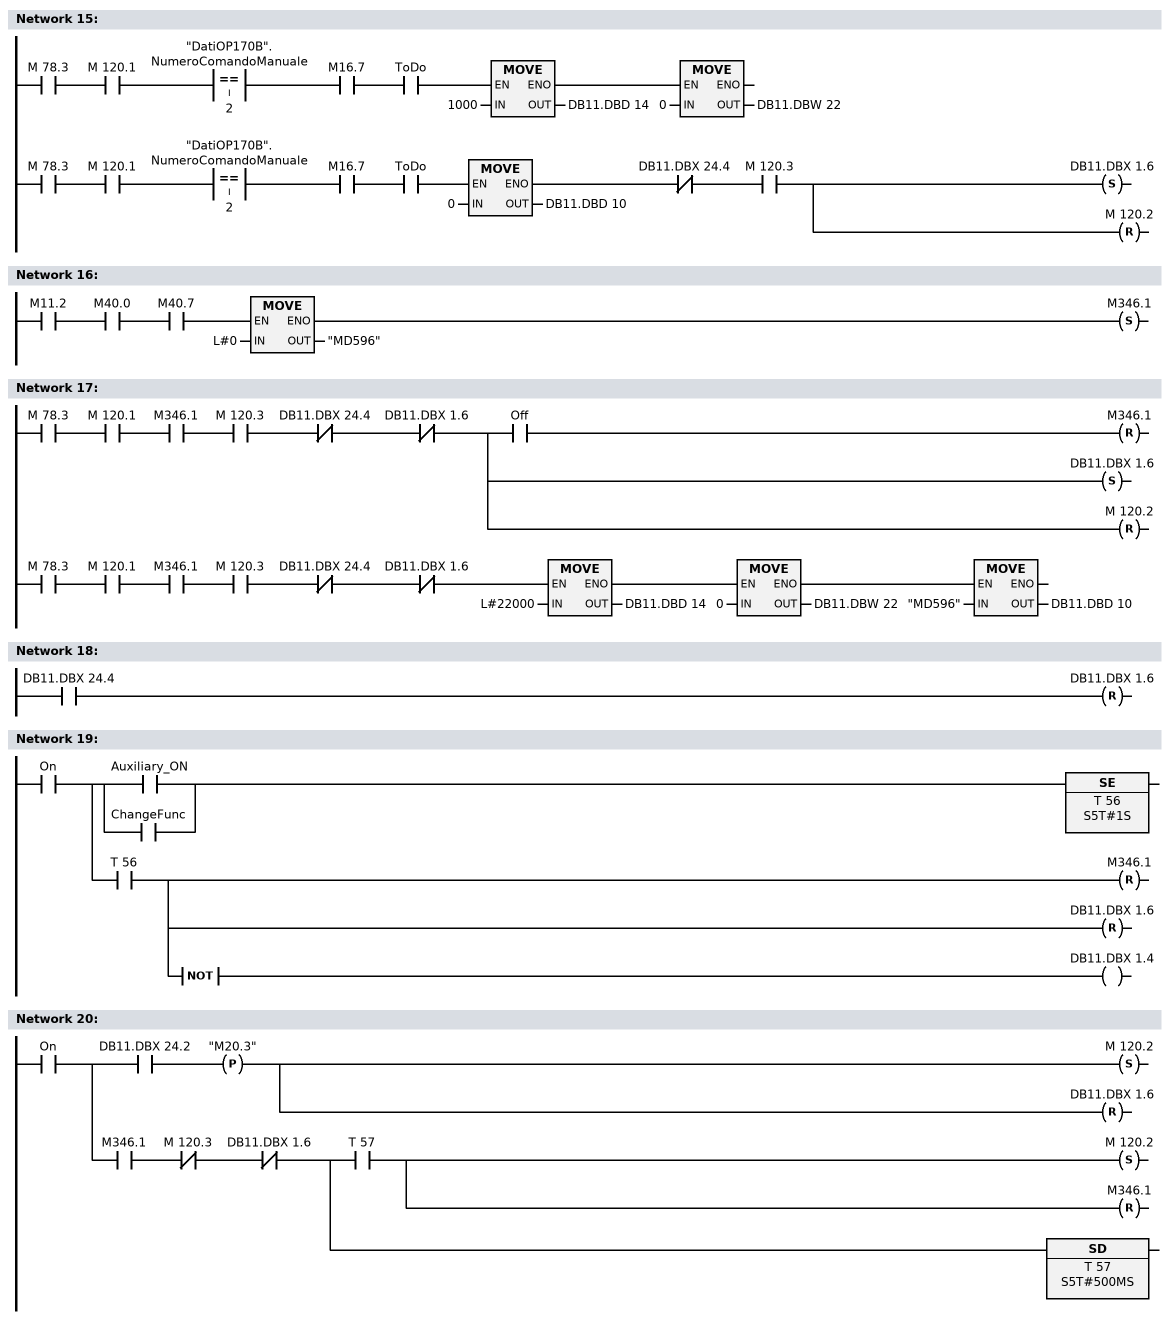
[picture p48: FC - AUTOMATIC networks 15-20]
NETWORK
TITLE =
      A     M 78.3;
      A     M 120.1;
      A(;
      L     "DatiOP170B".NumeroComandoManuale;
      L     2;
      ==I;
      );
      A     "M16.7";
      =     L 21.0;
      A(;
      A     L 21.0;
      A     "ToDo";
      JNB   M012;
      L     1000;
      T     DB11.DBD 14;
      SET;
      SAVE;
      CLR;
M012: A     BR;
      );
      JNB   M013;
      L     0;
      T     DB11.DBW 22;
M013: NOP   0;
      A(;
      A     L 21.0;
      A     "ToDo";
      JNB   M014;
      L     0;
      T     DB11.DBD 10;
      SET;
      SAVE;
      CLR;
M014: A     BR;
      );
      AN    DB11.DBX 24.4;
      A     M 120.3;
      S     DB11.DBX 1.6;
      R     M 120.2;
NETWORK
TITLE =
      A     "M11.2";
      A     "M40.0";
      A     "M40.7";
      JNB   M015;
      L     L#0;
      T     "MD596";
      SET;
      SAVE;
      CLR;
M015: A     BR;
      S     "M346.1";
NETWORK
TITLE =
      A     M 78.3;
      A     M 120.1;
      A     "M346.1";
      A     M 120.3;
      AN    DB11.DBX 24.4;
      AN    DB11.DBX 1.6;
      =     L 21.0;
      A(;
      A(;
      A     L 21.0;
      JNB   M016;
      L     L#22000;
      T     DB11.DBD 14;
      SET;
      SAVE;
      CLR;
M016: A     BR;
      );
      JNB   M017;
      L     0;
      T     DB11.DBW 22;
      SET;
      SAVE;
      CLR;
M017: A     BR;
      );
      JNB   M018;
      L     "MD596";
      T     DB11.DBD 10;
M018: NOP   0;
      A     L 21.0;
      A     "Off";
      R     "M346.1";
      A     L 21.0;
      BLD   102;
      S     DB11.DBX 1.6;
      A     L 21.0;
      BLD   102;
      R     M 120.2;
NETWORK
TITLE =
      A     DB11.DBX 24.4;
      R     DB11.DBX 1.6;
NETWORK
TITLE =
      A     "On";
      =     L 21.0;
      A     L 21.0;
      A(;
      O     "Auxiliary_ON";
      O     "ChangeFunc";
      );
      L     S5T#1S;
      SE    T 56;
      A     L 21.0;
      A     T 56;
      =     L 21.1;
      A     L 21.1;
      BLD   102;
      R     "M346.1";
      A     L 21.1;
      BLD   102;
      R     DB11.DBX 1.6;
      A     L 21.1;
      NOT;
      =     DB11.DBX 1.4;
NETWORK
TITLE =
      A     "On";
      =     L 21.0;
      A     L 21.0;
      A     DB11.DBX 24.2;
      FP    "M20.3";
      S     M 120.2;
      R     DB11.DBX 1.6;
      A     L 21.0;
      A     "M346.1";
      AN    M 120.3;
      AN    DB11.DBX 1.6;
      =     L 21.1;
      A     L 21.1;
      A     T 57;
      S     M 120.2;
      R     "M346.1";
      A     L 21.1;
      BLD   102;
      L     S5T#500MS;
      SD    T 57;
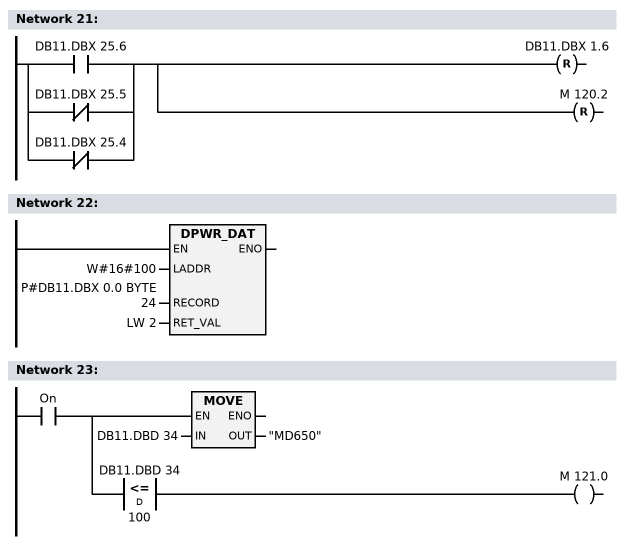
NETWORK
TITLE =
      O     DB11.DBX 25.6;
      ON    DB11.DBX 25.5;
      ON    DB11.DBX 25.4;
      R     DB11.DBX 1.6;
      R     M 120.2;
NETWORK
TITLE =
      CALL  "DPWR_DAT" (
           LADDR                    := W#16#100,
           RECORD                   := P#DB11.DBX 0.0 BYTE 24,
           RET_VAL                  := LW 2);
      NOP   0;
NETWORK
TITLE =
      A     "On";
      =     L 20.0;
      A     L 20.0;
      JNB   M019;
      L     DB11.DBD 34;
      T     "MD650";
M019: NOP   0;
      A     L 20.0;
      A(;
      L     DB11.DBD 34;
      L     100;
      <=D;
      );
      =     M 121.0;
END_FUNCTION

FUNCTION FC 25 : VOID
VERSION : 0.1
BEGIN
// (block stored without names or comments; labels and parameter names are numbered)
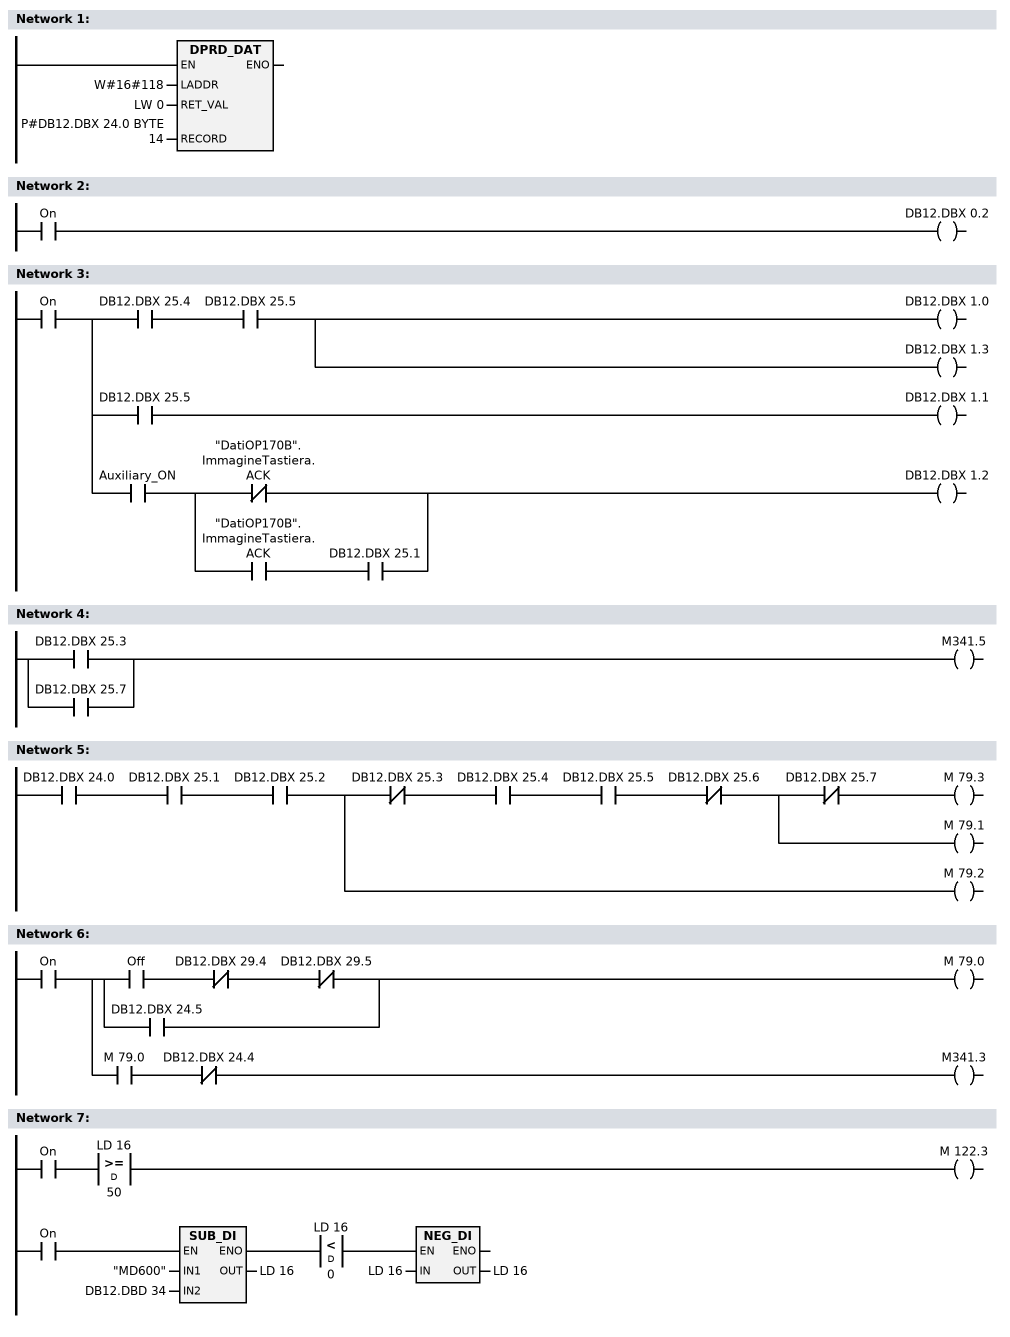
NETWORK
TITLE =
      CALL  "DPRD_DAT" (
           LADDR                    := W#16#118,
           RET_VAL                  := LW 0,
           RECORD                   := P#DB12.DBX 24.0 BYTE 14);
      NOP   0;
NETWORK
TITLE =
      A     "On";
      =     DB12.DBX 0.2;
NETWORK
TITLE =
      A     "On";
      =     L 21.0;
      A     L 21.0;
      A     DB12.DBX 25.4;
      A     DB12.DBX 25.5;
      =     DB12.DBX 1.0;
      =     DB12.DBX 1.3;
      A     L 21.0;
      A     DB12.DBX 25.5;
      =     DB12.DBX 1.1;
      A     L 21.0;
      A     "Auxiliary_ON";
      A(;
      ON    "DatiOP170B".ImmagineTastiera.ACK;
      O;
      A     "DatiOP170B".ImmagineTastiera.ACK;
      A     DB12.DBX 25.1;
      );
      =     DB12.DBX 1.2;
NETWORK
TITLE =
      O     DB12.DBX 25.3;
      O     DB12.DBX 25.7;
      =     "M341.5";
NETWORK
TITLE =
      A     DB12.DBX 24.0;
      A     DB12.DBX 25.1;
      A     DB12.DBX 25.2;
      =     L 21.0;
      A     L 21.0;
      AN    DB12.DBX 25.3;
      A     DB12.DBX 25.4;
      A     DB12.DBX 25.5;
      AN    DB12.DBX 25.6;
      =     L 21.1;
      A     L 21.1;
      AN    DB12.DBX 25.7;
      =     M 79.3;
      A     L 21.1;
      BLD   102;
      =     M 79.1;
      A     L 21.0;
      BLD   102;
      =     M 79.2;
NETWORK
TITLE =
      A     "On";
      =     L 21.0;
      A     L 21.0;
      A(;
      A     "Off";
      AN    DB12.DBX 29.4;
      AN    DB12.DBX 29.5;
      O     DB12.DBX 24.5;
      );
      =     M 79.0;
      A     L 21.0;
      A     M 79.0;
      AN    DB12.DBX 24.4;
      =     "M341.3";
NETWORK
TITLE =
      A     "On";
      =     L 20.0;
      A(;
      A     L 20.0;
      JNB   M001;
      L     "MD600";
      L     DB12.DBD 34;
      -D;
      T     LD 16;
      AN    OV;
      SAVE;
      CLR;
M001: A     BR;
      );
      A(;
      L     LD 16;
      L     0;
      <D;
      );
      JNB   M002;
      L     LD 16;
      NEGD;
      T     LD 16;
M002: NOP   0;
      A     L 20.0;
      A(;
      L     LD 16;
      L     50;
      >=D;
      );
      =     M 122.3;
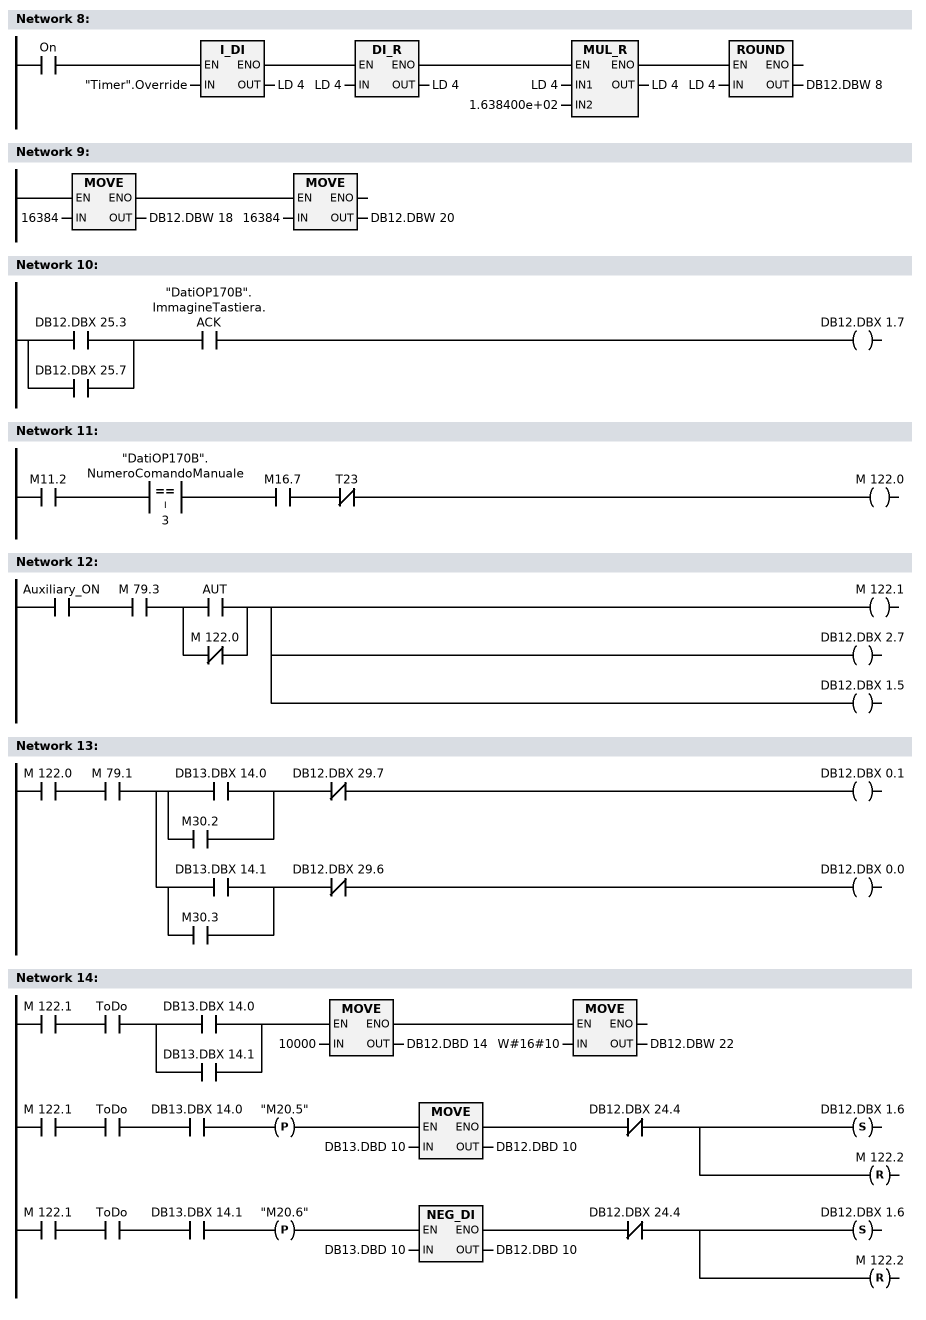
NETWORK
TITLE =
      A(;
      A(;
      A(;
      A     "On";
      JNB   M003;
      L     "Timer".Override;
      ITD;
      T     LD 4;
      SET;
      SAVE;
      CLR;
M003: A     BR;
      );
      JNB   M004;
      L     LD 4;
      DTR;
      T     LD 4;
      SET;
      SAVE;
      CLR;
M004: A     BR;
      );
      JNB   M005;
      L     LD 4;
      L     1.638400e+02;
      *R;
      T     LD 4;
      AN    OV;
      SAVE;
      CLR;
M005: A     BR;
      );
      JNB   M006;
      L     LD 4;
      RND;
      T     DB12.DBW 8;
M006: NOP   0;
NETWORK
TITLE =
      A(;
      L     16384;
      T     DB12.DBW 18;
      SET;
      SAVE;
      CLR;
      A     BR;
      );
      JNB   M007;
      L     16384;
      T     DB12.DBW 20;
M007: NOP   0;
NETWORK
TITLE =
      A(;
      O     DB12.DBX 25.3;
      O     DB12.DBX 25.7;
      );
      A     "DatiOP170B".ImmagineTastiera.ACK;
      =     DB12.DBX 1.7;
NETWORK
TITLE =
      A     "M11.2";
      A(;
      L     "DatiOP170B".NumeroComandoManuale;
      L     3;
      ==I;
      );
      A     "M16.7";
      AN    "T23";
      =     M 122.0;
NETWORK
TITLE =
      A     "Auxiliary_ON";
      A     M 79.3;
      A(;
      O     "AUT";
      ON    M 122.0;
      );
      =     M 122.1;
      =     DB12.DBX 2.7;
      =     DB12.DBX 1.5;
NETWORK
TITLE =
      A     M 122.0;
      A     M 79.1;
      =     L 21.0;
      A     L 21.0;
      A(;
      O     DB13.DBX 14.0;
      O     "M30.2";
      );
      AN    DB12.DBX 29.7;
      =     DB12.DBX 0.1;
      A     L 21.0;
      A(;
      O     DB13.DBX 14.1;
      O     "M30.3";
      );
      AN    DB12.DBX 29.6;
      =     DB12.DBX 0.0;
NETWORK
TITLE =
      A     M 122.1;
      A     "ToDo";
      =     L 21.0;
      A(;
      A     L 21.0;
      A(;
      O     DB13.DBX 14.0;
      O     DB13.DBX 14.1;
      );
      JNB   M008;
      L     10000;
      T     DB12.DBD 14;
      SET;
      SAVE;
      CLR;
M008: A     BR;
      );
      JNB   M009;
      L     W#16#10;
      T     DB12.DBW 22;
M009: NOP   0;
      A(;
      A     L 21.0;
      A     DB13.DBX 14.0;
      FP    "M20.5";
      JNB   M010;
      L     DB13.DBD 10;
      T     DB12.DBD 10;
      SET;
      SAVE;
      CLR;
M010: A     BR;
      );
      AN    DB12.DBX 24.4;
      S     DB12.DBX 1.6;
      R     M 122.2;
      A(;
      A     L 21.0;
      A     DB13.DBX 14.1;
      FP    "M20.6";
      JNB   M011;
      L     DB13.DBD 10;
      NEGD;
      T     DB12.DBD 10;
      AN    OV;
      SAVE;
      CLR;
M011: A     BR;
      );
      AN    DB12.DBX 24.4;
      S     DB12.DBX 1.6;
      R     M 122.2;
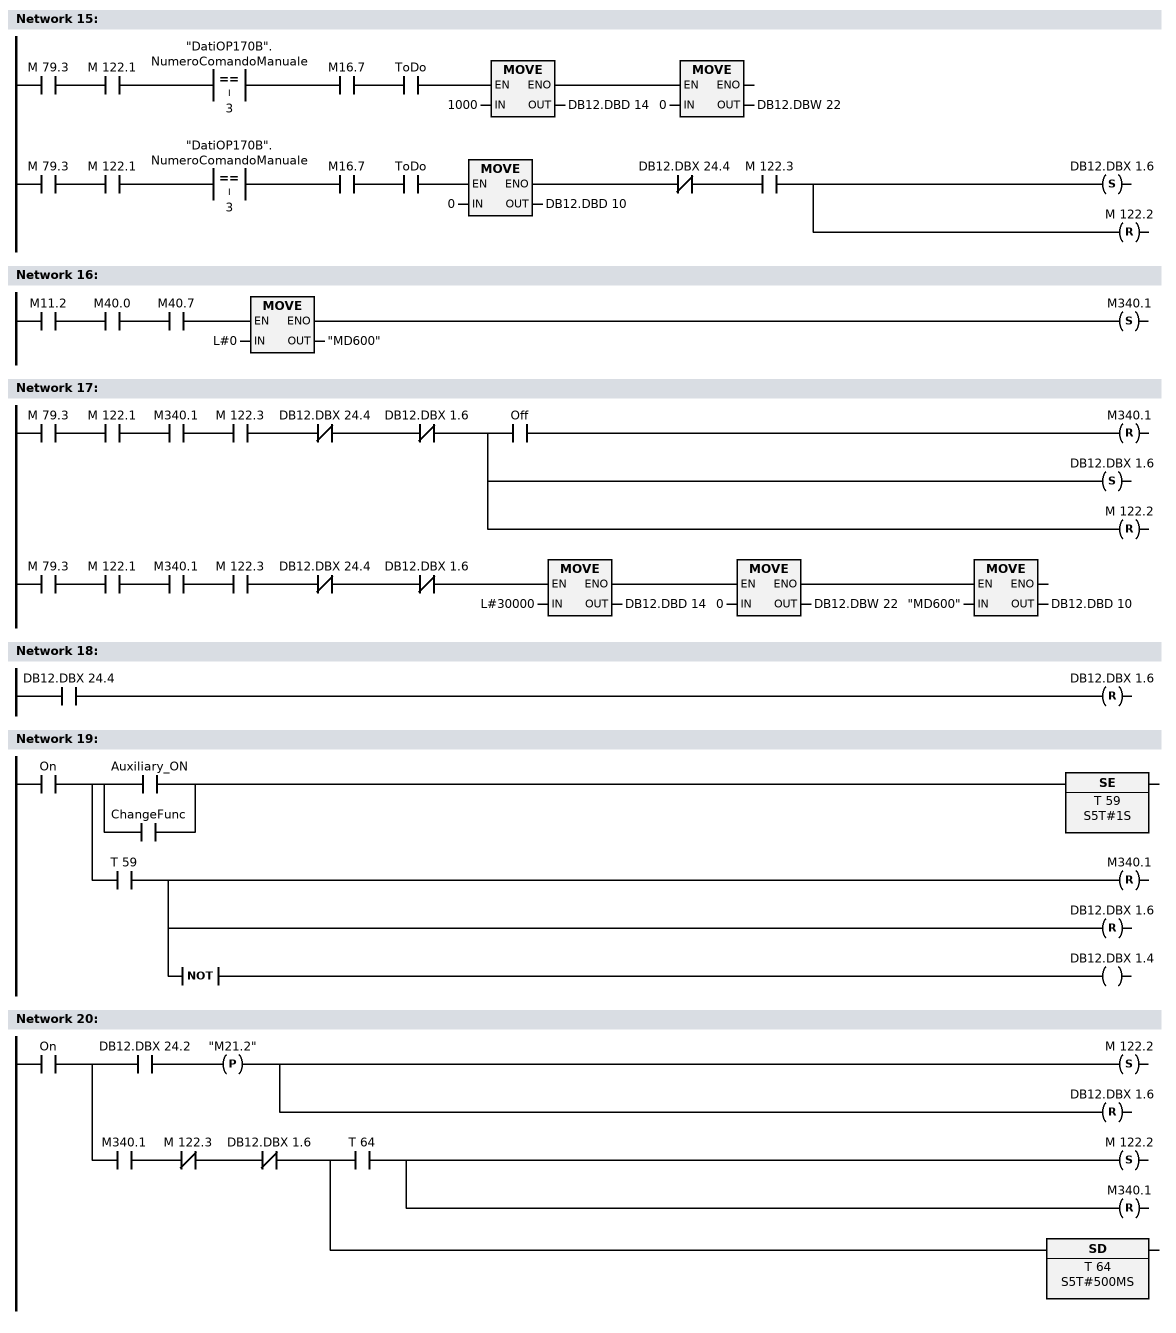
NETWORK
TITLE =
      A     M 79.3;
      A     M 122.1;
      A(;
      L     "DatiOP170B".NumeroComandoManuale;
      L     3;
      ==I;
      );
      A     "M16.7";
      =     L 21.0;
      A(;
      A     L 21.0;
      A     "ToDo";
      JNB   M012;
      L     1000;
      T     DB12.DBD 14;
      SET;
      SAVE;
      CLR;
M012: A     BR;
      );
      JNB   M013;
      L     0;
      T     DB12.DBW 22;
M013: NOP   0;
      A(;
      A     L 21.0;
      A     "ToDo";
      JNB   M014;
      L     0;
      T     DB12.DBD 10;
      SET;
      SAVE;
      CLR;
M014: A     BR;
      );
      AN    DB12.DBX 24.4;
      A     M 122.3;
      S     DB12.DBX 1.6;
      R     M 122.2;
NETWORK
TITLE =
      A     "M11.2";
      A     "M40.0";
      A     "M40.7";
      JNB   M015;
      L     L#0;
      T     "MD600";
      SET;
      SAVE;
      CLR;
M015: A     BR;
      S     "M340.1";
NETWORK
TITLE =
      A     M 79.3;
      A     M 122.1;
      A     "M340.1";
      A     M 122.3;
      AN    DB12.DBX 24.4;
      AN    DB12.DBX 1.6;
      =     L 21.0;
      A(;
      A(;
      A     L 21.0;
      JNB   M016;
      L     L#30000;
      T     DB12.DBD 14;
      SET;
      SAVE;
      CLR;
M016: A     BR;
      );
      JNB   M017;
      L     0;
      T     DB12.DBW 22;
      SET;
      SAVE;
      CLR;
M017: A     BR;
      );
      JNB   M018;
      L     "MD600";
      T     DB12.DBD 10;
M018: NOP   0;
      A     L 21.0;
      A     "Off";
      R     "M340.1";
      A     L 21.0;
      BLD   102;
      S     DB12.DBX 1.6;
      A     L 21.0;
      BLD   102;
      R     M 122.2;
NETWORK
TITLE =
      A     DB12.DBX 24.4;
      R     DB12.DBX 1.6;
NETWORK
TITLE =
      A     "On";
      =     L 21.0;
      A     L 21.0;
      A(;
      O     "Auxiliary_ON";
      O     "ChangeFunc";
      );
      L     S5T#1S;
      SE    T 59;
      A     L 21.0;
      A     T 59;
      =     L 21.1;
      A     L 21.1;
      BLD   102;
      R     "M340.1";
      A     L 21.1;
      BLD   102;
      R     DB12.DBX 1.6;
      A     L 21.1;
      NOT;
      =     DB12.DBX 1.4;
NETWORK
TITLE =
      A     "On";
      =     L 21.0;
      A     L 21.0;
      A     DB12.DBX 24.2;
      FP    "M21.2";
      S     M 122.2;
      R     DB12.DBX 1.6;
      A     L 21.0;
      A     "M340.1";
      AN    M 122.3;
      AN    DB12.DBX 1.6;
      =     L 21.1;
      A     L 21.1;
      A     T 64;
      S     M 122.2;
      R     "M340.1";
      A     L 21.1;
      BLD   102;
      L     S5T#500MS;
      SD    T 64;
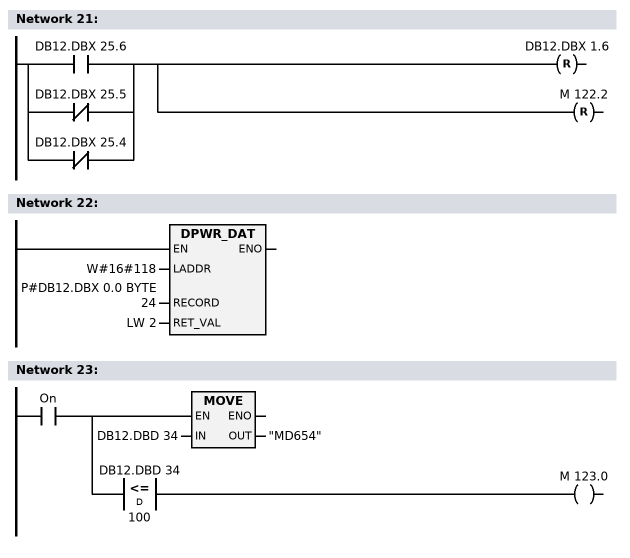
NETWORK
TITLE =
      O     DB12.DBX 25.6;
      ON    DB12.DBX 25.5;
      ON    DB12.DBX 25.4;
      R     DB12.DBX 1.6;
      R     M 122.2;
NETWORK
TITLE =
      CALL  "DPWR_DAT" (
           LADDR                    := W#16#118,
           RECORD                   := P#DB12.DBX 0.0 BYTE 24,
           RET_VAL                  := LW 2);
      NOP   0;
NETWORK
TITLE =
      A     "On";
      =     L 20.0;
      A     L 20.0;
      JNB   M019;
      L     DB12.DBD 34;
      T     "MD654";
M019: NOP   0;
      A     L 20.0;
      A(;
      L     DB12.DBD 34;
      L     100;
      <=D;
      );
      =     M 123.0;
END_FUNCTION

FUNCTION "FC50 - TEACH-IN" : VOID	// FC 50
VERSION : 0.1
VAR_TEMP
  TEMP0 : DINT ;
  TEMP1 : DINT ;
END_VAR
BEGIN
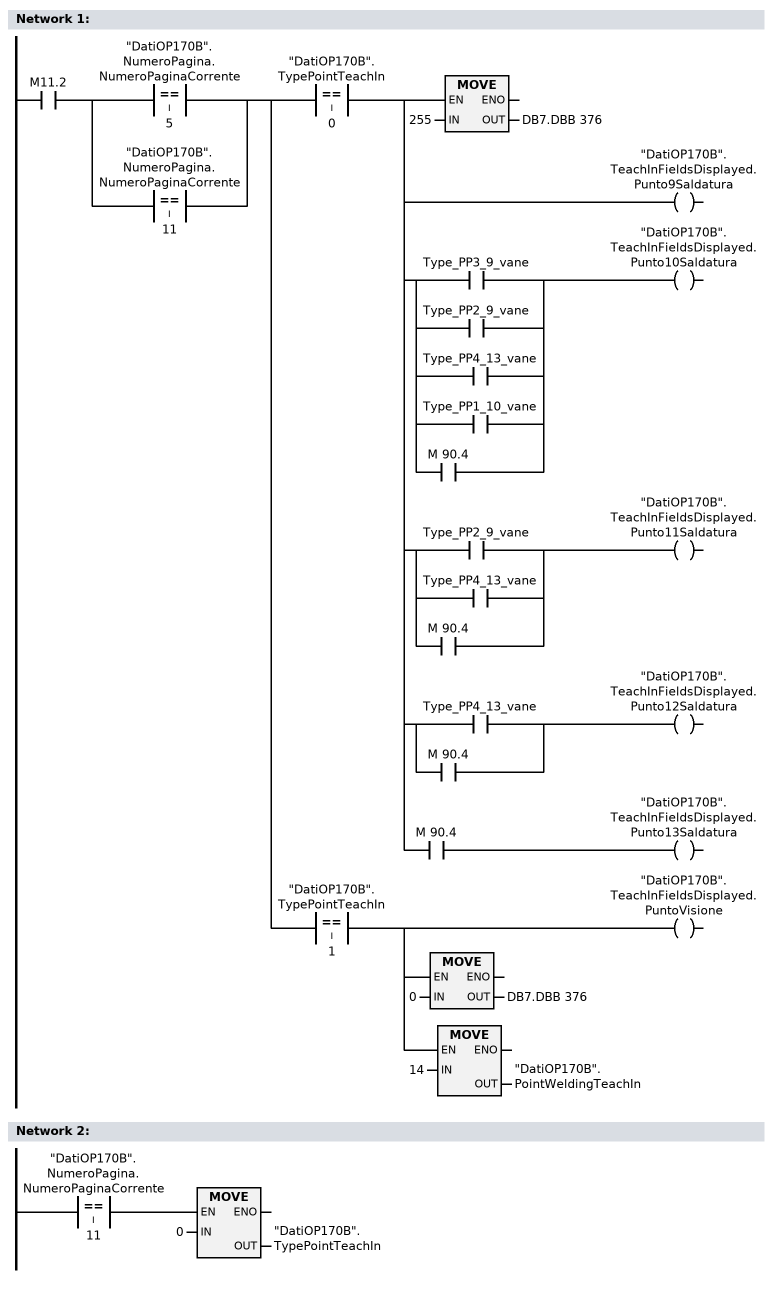
NETWORK
TITLE =
      A     "M11.2";
      A(;
      O(;
      L     "DatiOP170B".NumeroPagina.NumeroPaginaCorrente;
      L     5;
      ==I;
      );
      O(;
      L     "DatiOP170B".NumeroPagina.NumeroPaginaCorrente;
      L     11;
      ==I;
      );
      );
      =     L 8.0;
      A     L 8.0;
      A(;
      L     "DatiOP170B".TypePointTeachIn;
      L     0;
      ==I;
      );
      =     L 8.1;
      A     L 8.1;
      JNB   _001;
      L     255;
      T     DB7.DBB 376;
_001: NOP   0;
      A     L 8.1;
      BLD   102;
      =     "DatiOP170B".TeachInFieldsDisplayed.Punto9Saldatura;
      A     L 8.1;
      A(;
      O     "Type_PP3_9_vane";
      O     "Type_PP2_9_vane";
      O     "Type_PP4_13_vane";
      O     "Type_PP1_10_vane";
      O     M 90.4;
      );
      =     "DatiOP170B".TeachInFieldsDisplayed.Punto10Saldatura;
      A     L 8.1;
      A(;
      O     "Type_PP2_9_vane";
      O     "Type_PP4_13_vane";
      O     M 90.4;
      );
      =     "DatiOP170B".TeachInFieldsDisplayed.Punto11Saldatura;
      A     L 8.1;
      A(;
      O     "Type_PP4_13_vane";
      O     M 90.4;
      );
      =     "DatiOP170B".TeachInFieldsDisplayed.Punto12Saldatura;
      A     L 8.1;
      A     M 90.4;
      =     "DatiOP170B".TeachInFieldsDisplayed.Punto13Saldatura;
      A     L 8.0;
      A(;
      L     "DatiOP170B".TypePointTeachIn;
      L     1;
      ==I;
      );
      =     L 8.1;
      A     L 8.1;
      BLD   102;
      =     "DatiOP170B".TeachInFieldsDisplayed.PuntoVisione;
      A     L 8.1;
      JNB   _002;
      L     0;
      T     DB7.DBB 376;
_002: NOP   0;
      A     L 8.1;
      JNB   _003;
      L     14;
      T     "DatiOP170B".PointWeldingTeachIn;
_003: NOP   0;
NETWORK
TITLE =
      A(;
      L     "DatiOP170B".NumeroPagina.NumeroPaginaCorrente;
      L     11;
      ==I;
      );
      JNB   _004;
      L     0;
      T     "DatiOP170B".TypePointTeachIn;
_004: NOP   0;
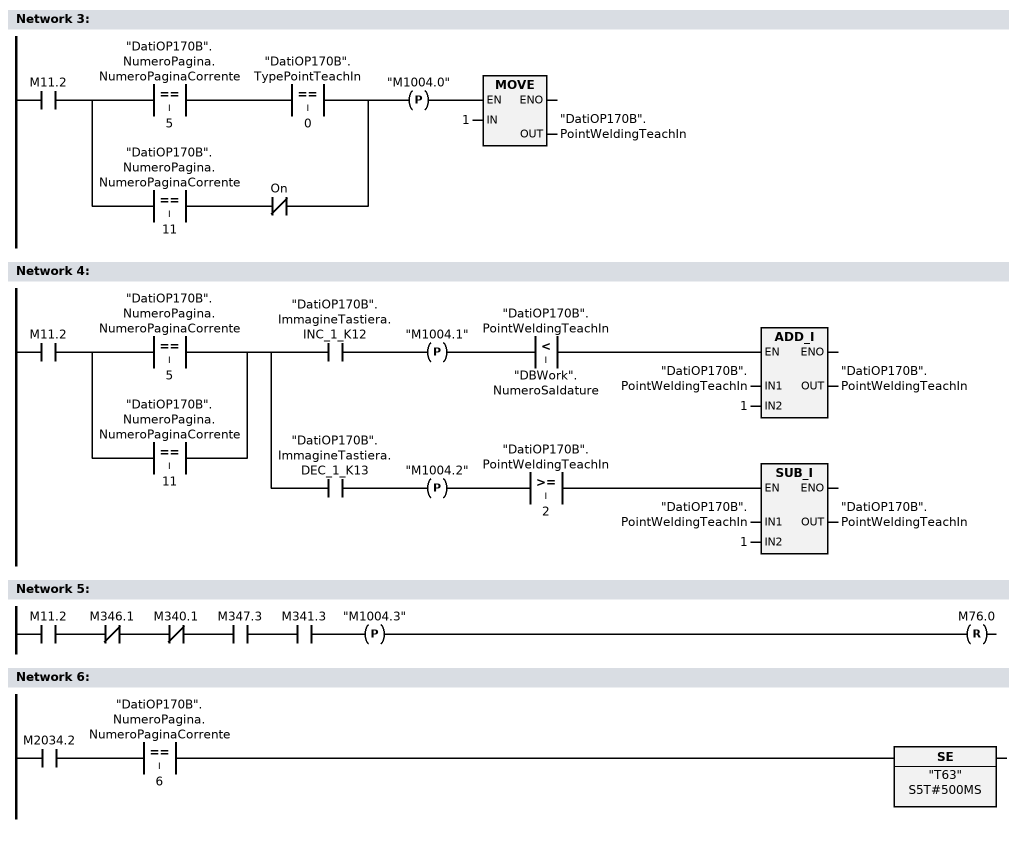
NETWORK
TITLE =
      A     "M11.2";
      A(;
      A(;
      L     "DatiOP170B".NumeroPagina.NumeroPaginaCorrente;
      L     5;
      ==I;
      );
      A(;
      L     "DatiOP170B".TypePointTeachIn;
      L     0;
      ==I;
      );
      O;
      A(;
      L     "DatiOP170B".NumeroPagina.NumeroPaginaCorrente;
      L     11;
      ==I;
      );
      AN    "On";
      );
      FP    "M1004.0";
      JNB   _005;
      L     1;
      T     "DatiOP170B".PointWeldingTeachIn;
_005: NOP   0;
NETWORK
TITLE =
      A     "M11.2";
      A(;
      O(;
      L     "DatiOP170B".NumeroPagina.NumeroPaginaCorrente;
      L     5;
      ==I;
      );
      O(;
      L     "DatiOP170B".NumeroPagina.NumeroPaginaCorrente;
      L     11;
      ==I;
      );
      );
      =     L 8.0;
      A     L 8.0;
      A     "DatiOP170B".ImmagineTastiera.INC_1_K12;
      FP    "M1004.1";
      A(;
      L     "DatiOP170B".PointWeldingTeachIn;
      L     "DBWork".NumeroSaldature;
      <I;
      );
      JNB   _006;
      L     "DatiOP170B".PointWeldingTeachIn;
      L     1;
      +I;
      T     "DatiOP170B".PointWeldingTeachIn;
_006: NOP   0;
      A     L 8.0;
      A     "DatiOP170B".ImmagineTastiera.DEC_1_K13;
      FP    "M1004.2";
      A(;
      L     "DatiOP170B".PointWeldingTeachIn;
      L     2;
      >=I;
      );
      JNB   _007;
      L     "DatiOP170B".PointWeldingTeachIn;
      L     1;
      -I;
      T     "DatiOP170B".PointWeldingTeachIn;
_007: NOP   0;
NETWORK
TITLE =
      A     "M11.2";
      AN    "M346.1";
      AN    "M340.1";
      A     "M347.3";
      A     "M341.3";
      FP    "M1004.3";
      R     "M76.0";
NETWORK
TITLE =
      A     "M2034.2";
      A(;
      L     "DatiOP170B".NumeroPagina.NumeroPaginaCorrente;
      L     6;
      ==I;
      );
      L     S5T#500MS;
      SE    "T63";
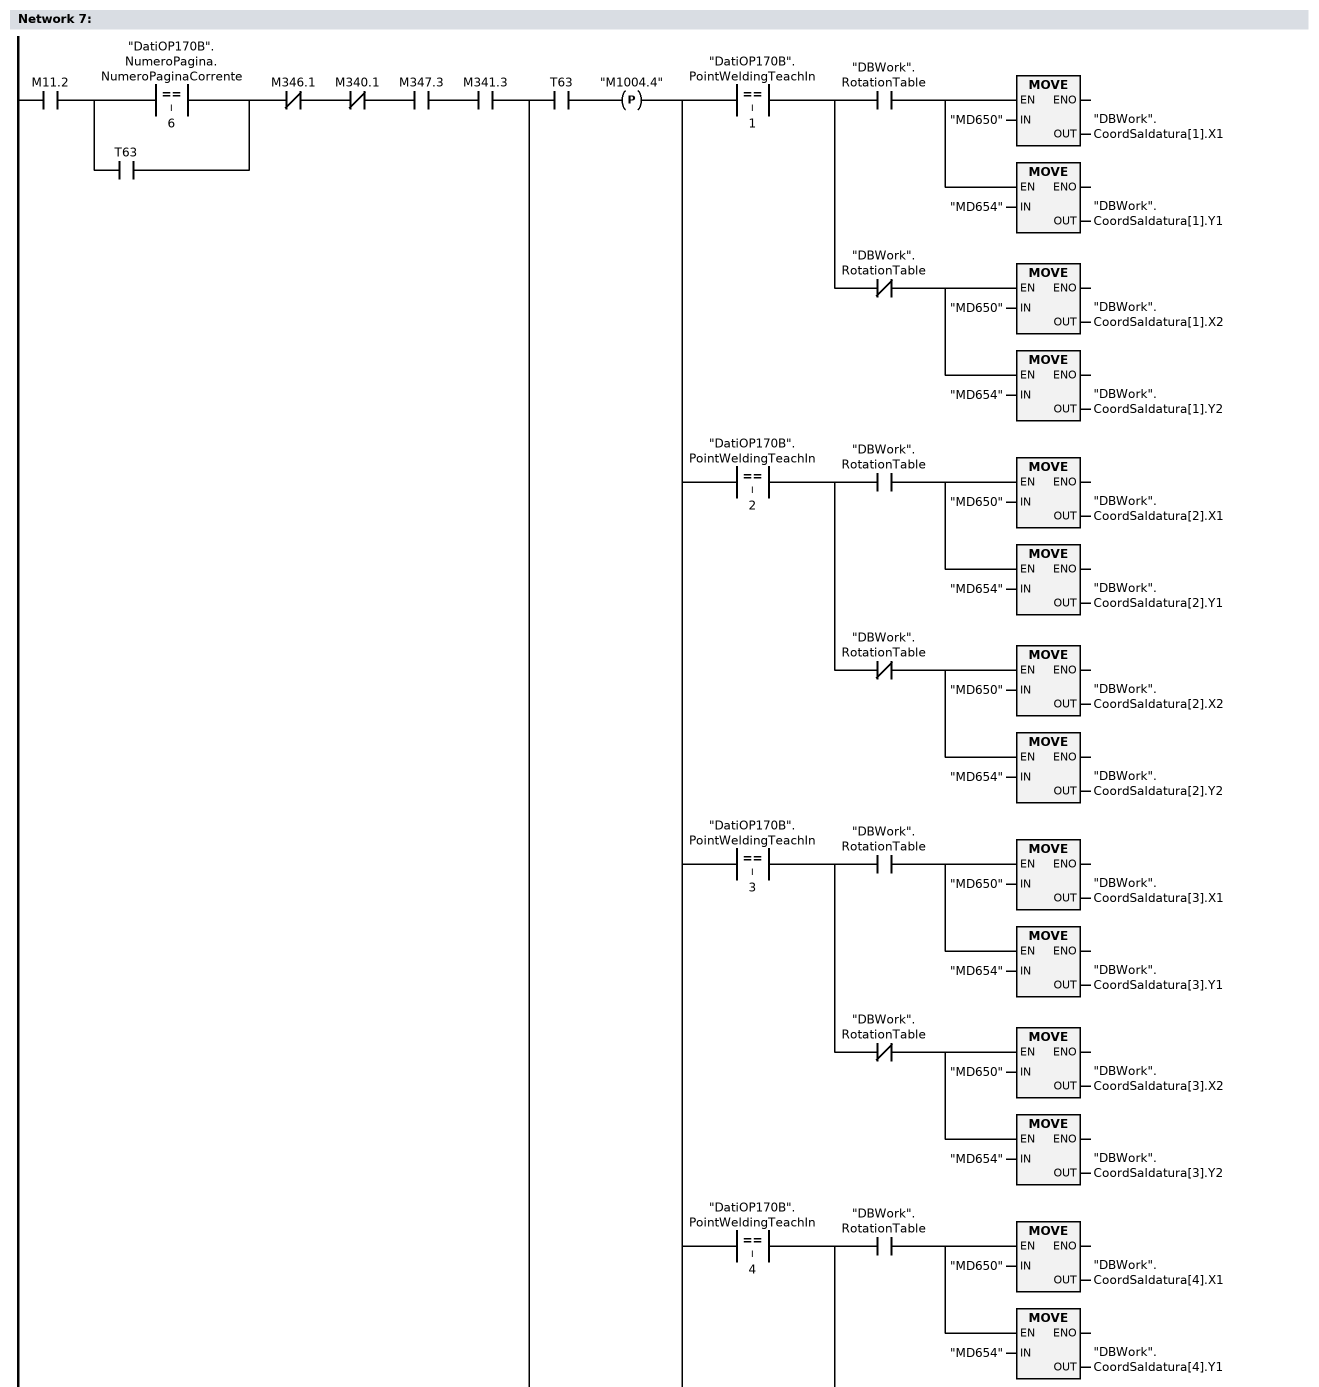
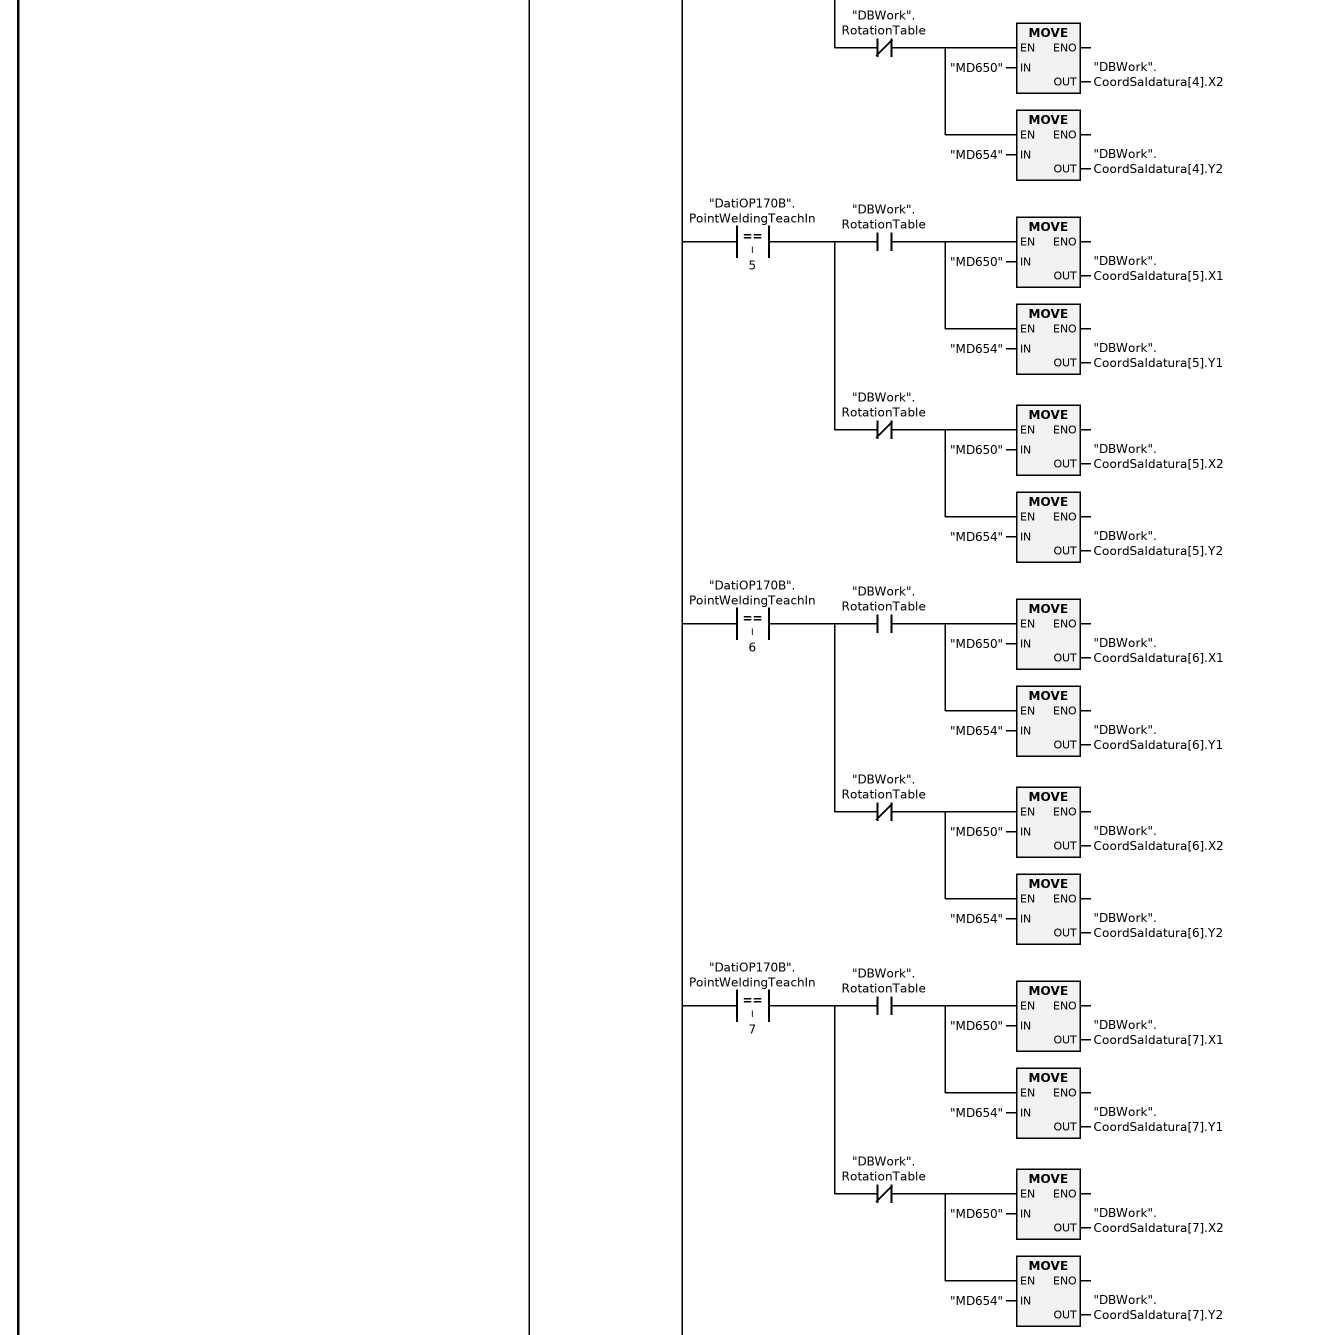
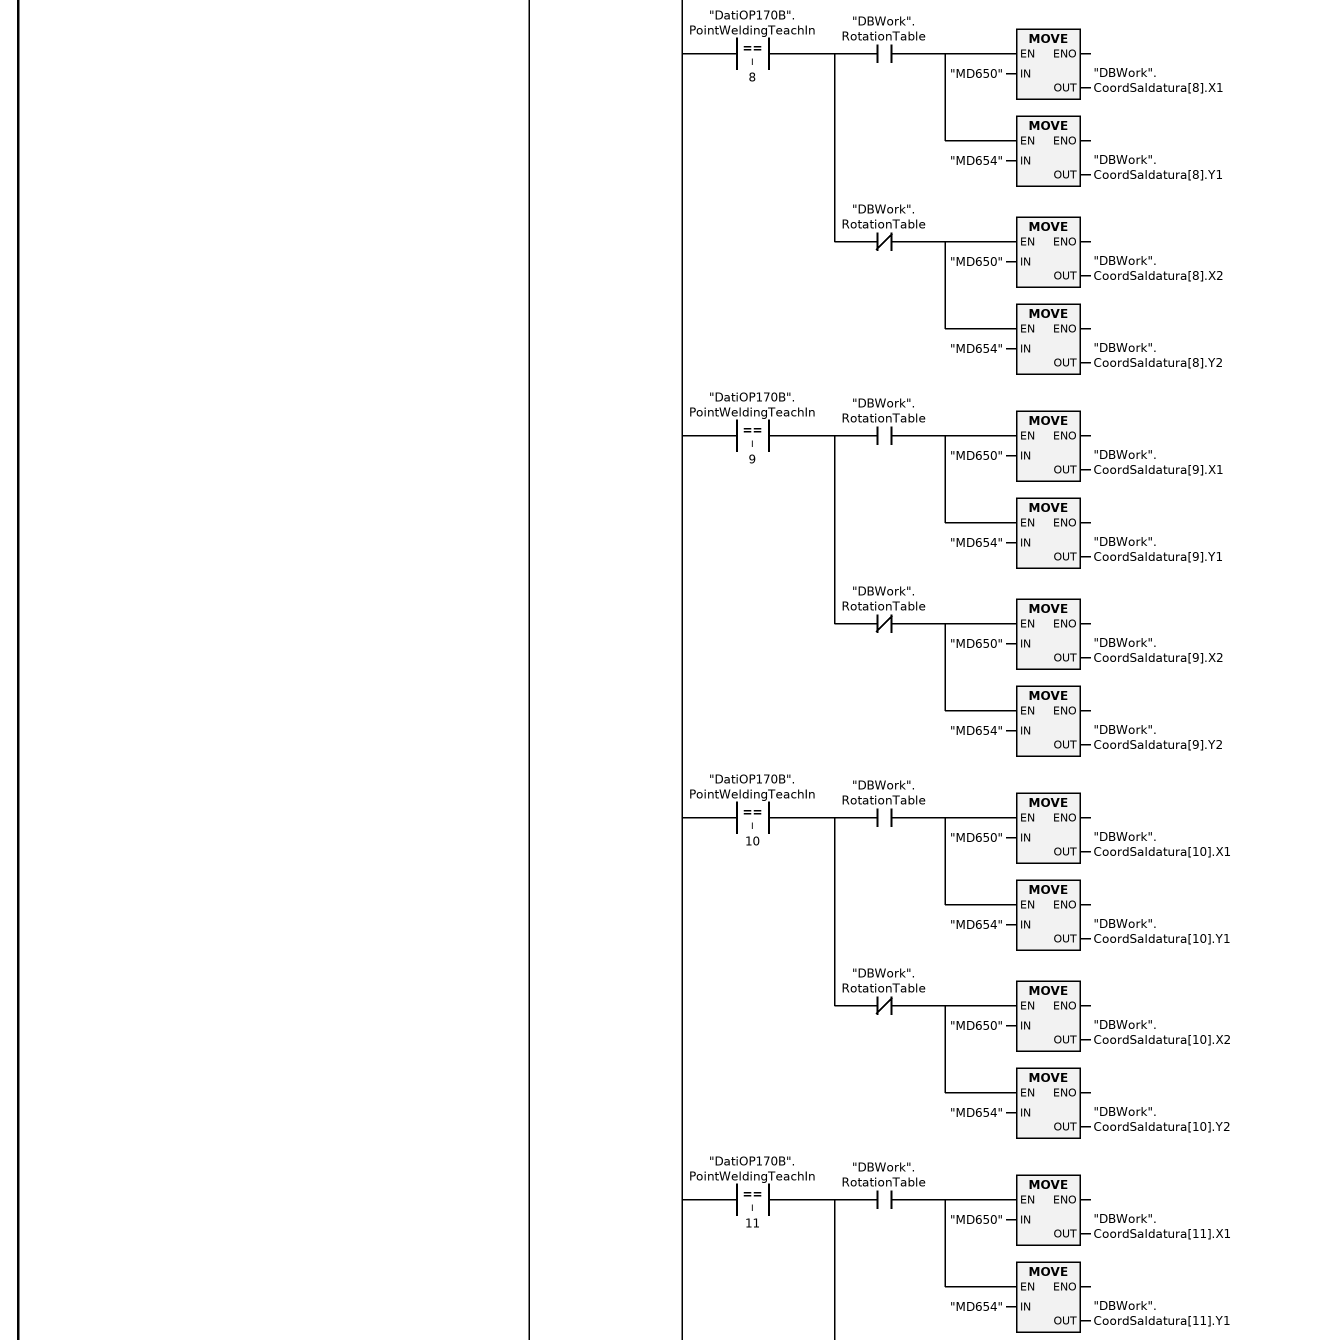
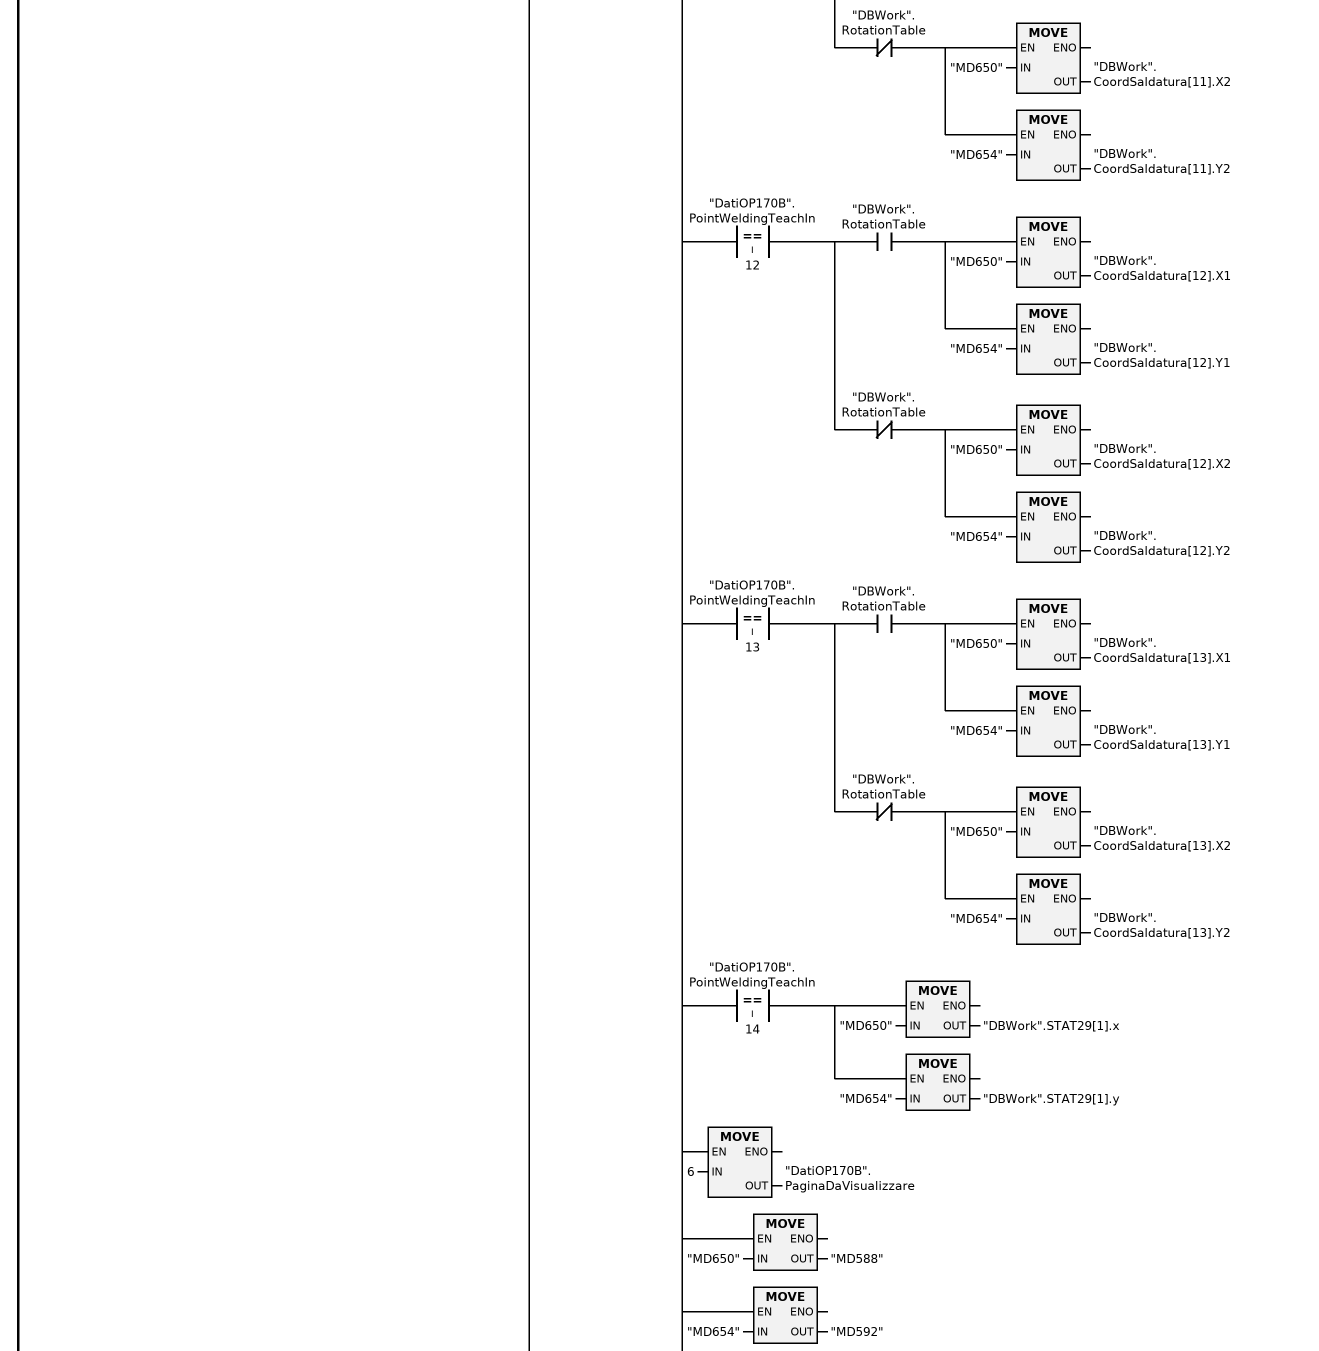
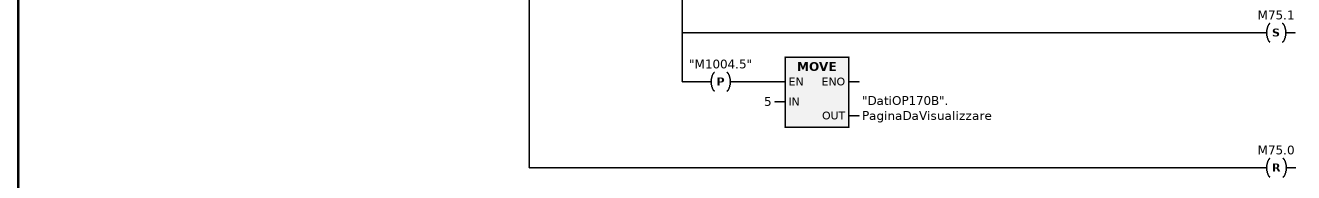
NETWORK
TITLE =
      A     "M11.2";
      A(;
      O(;
      L     "DatiOP170B".NumeroPagina.NumeroPaginaCorrente;
      L     6;
      ==I;
      );
      O     "T63";
      );
      AN    "M346.1";
      AN    "M340.1";
      A     "M347.3";
      A     "M341.3";
      =     L 8.0;
      A     L 8.0;
      A     "T63";
      FP    "M1004.4";
      =     L 8.1;
      A     L 8.1;
      A(;
      L     "DatiOP170B".PointWeldingTeachIn;
      L     1;
      ==I;
      );
      =     L 8.2;
      A     L 8.2;
      A     "DBWork".RotationTable;
      =     L 8.3;
      A     L 8.3;
      JNB   _008;
      L     "MD650";
      T     "DBWork".CoordSaldatura[1].X1;
_008: NOP   0;
      A     L 8.3;
      JNB   _009;
      L     "MD654";
      T     "DBWork".CoordSaldatura[1].Y1;
_009: NOP   0;
      A     L 8.2;
      AN    "DBWork".RotationTable;
      =     L 8.3;
      A     L 8.3;
      JNB   _00a;
      L     "MD650";
      T     "DBWork".CoordSaldatura[1].X2;
_00a: NOP   0;
      A     L 8.3;
      JNB   _00b;
      L     "MD654";
      T     "DBWork".CoordSaldatura[1].Y2;
_00b: NOP   0;
      A     L 8.1;
      A(;
      L     "DatiOP170B".PointWeldingTeachIn;
      L     2;
      ==I;
      );
      =     L 8.2;
      A     L 8.2;
      A     "DBWork".RotationTable;
      =     L 8.3;
      A     L 8.3;
      JNB   _00c;
      L     "MD650";
      T     "DBWork".CoordSaldatura[2].X1;
_00c: NOP   0;
      A     L 8.3;
      JNB   _00d;
      L     "MD654";
      T     "DBWork".CoordSaldatura[2].Y1;
_00d: NOP   0;
      A     L 8.2;
      AN    "DBWork".RotationTable;
      =     L 8.3;
      A     L 8.3;
      JNB   _00e;
      L     "MD650";
      T     "DBWork".CoordSaldatura[2].X2;
_00e: NOP   0;
      A     L 8.3;
      JNB   _00f;
      L     "MD654";
      T     "DBWork".CoordSaldatura[2].Y2;
_00f: NOP   0;
      A     L 8.1;
      A(;
      L     "DatiOP170B".PointWeldingTeachIn;
      L     3;
      ==I;
      );
      =     L 8.2;
      A     L 8.2;
      A     "DBWork".RotationTable;
      =     L 8.3;
      A     L 8.3;
      JNB   _010;
      L     "MD650";
      T     "DBWork".CoordSaldatura[3].X1;
_010: NOP   0;
      A     L 8.3;
      JNB   _011;
      L     "MD654";
      T     "DBWork".CoordSaldatura[3].Y1;
_011: NOP   0;
      A     L 8.2;
      AN    "DBWork".RotationTable;
      =     L 8.3;
      A     L 8.3;
      JNB   _012;
      L     "MD650";
      T     "DBWork".CoordSaldatura[3].X2;
_012: NOP   0;
      A     L 8.3;
      JNB   _013;
      L     "MD654";
      T     "DBWork".CoordSaldatura[3].Y2;
_013: NOP   0;
      A     L 8.1;
      A(;
      L     "DatiOP170B".PointWeldingTeachIn;
      L     4;
      ==I;
      );
      =     L 8.2;
      A     L 8.2;
      A     "DBWork".RotationTable;
      =     L 8.3;
      A     L 8.3;
      JNB   _014;
      L     "MD650";
      T     "DBWork".CoordSaldatura[4].X1;
_014: NOP   0;
      A     L 8.3;
      JNB   _015;
      L     "MD654";
      T     "DBWork".CoordSaldatura[4].Y1;
_015: NOP   0;
      A     L 8.2;
      AN    "DBWork".RotationTable;
      =     L 8.3;
      A     L 8.3;
      JNB   _016;
      L     "MD650";
      T     "DBWork".CoordSaldatura[4].X2;
_016: NOP   0;
      A     L 8.3;
      JNB   _017;
      L     "MD654";
      T     "DBWork".CoordSaldatura[4].Y2;
_017: NOP   0;
      A     L 8.1;
      A(;
      L     "DatiOP170B".PointWeldingTeachIn;
      L     5;
      ==I;
      );
      =     L 8.2;
      A     L 8.2;
      A     "DBWork".RotationTable;
      =     L 8.3;
      A     L 8.3;
      JNB   _018;
      L     "MD650";
      T     "DBWork".CoordSaldatura[5].X1;
_018: NOP   0;
      A     L 8.3;
      JNB   _019;
      L     "MD654";
      T     "DBWork".CoordSaldatura[5].Y1;
_019: NOP   0;
      A     L 8.2;
      AN    "DBWork".RotationTable;
      =     L 8.3;
      A     L 8.3;
      JNB   _01a;
      L     "MD650";
      T     "DBWork".CoordSaldatura[5].X2;
_01a: NOP   0;
      A     L 8.3;
      JNB   _01b;
      L     "MD654";
      T     "DBWork".CoordSaldatura[5].Y2;
_01b: NOP   0;
      A     L 8.1;
      A(;
      L     "DatiOP170B".PointWeldingTeachIn;
      L     6;
      ==I;
      );
      =     L 8.2;
      A     L 8.2;
      A     "DBWork".RotationTable;
      =     L 8.3;
      A     L 8.3;
      JNB   _01c;
      L     "MD650";
      T     "DBWork".CoordSaldatura[6].X1;
_01c: NOP   0;
      A     L 8.3;
      JNB   _01d;
      L     "MD654";
      T     "DBWork".CoordSaldatura[6].Y1;
_01d: NOP   0;
      A     L 8.2;
      AN    "DBWork".RotationTable;
      =     L 8.3;
      A     L 8.3;
      JNB   _01e;
      L     "MD650";
      T     "DBWork".CoordSaldatura[6].X2;
_01e: NOP   0;
      A     L 8.3;
      JNB   _01f;
      L     "MD654";
      T     "DBWork".CoordSaldatura[6].Y2;
_01f: NOP   0;
      A     L 8.1;
      A(;
      L     "DatiOP170B".PointWeldingTeachIn;
      L     7;
      ==I;
      );
      =     L 8.2;
      A     L 8.2;
      A     "DBWork".RotationTable;
      =     L 8.3;
      A     L 8.3;
      JNB   _020;
      L     "MD650";
      T     "DBWork".CoordSaldatura[7].X1;
_020: NOP   0;
      A     L 8.3;
      JNB   _021;
      L     "MD654";
      T     "DBWork".CoordSaldatura[7].Y1;
_021: NOP   0;
      A     L 8.2;
      AN    "DBWork".RotationTable;
      =     L 8.3;
      A     L 8.3;
      JNB   _022;
      L     "MD650";
      T     "DBWork".CoordSaldatura[7].X2;
_022: NOP   0;
      A     L 8.3;
      JNB   _023;
      L     "MD654";
      T     "DBWork".CoordSaldatura[7].Y2;
_023: NOP   0;
      A     L 8.1;
      A(;
      L     "DatiOP170B".PointWeldingTeachIn;
      L     8;
      ==I;
      );
      =     L 8.2;
      A     L 8.2;
      A     "DBWork".RotationTable;
      =     L 8.3;
      A     L 8.3;
      JNB   _024;
      L     "MD650";
      T     "DBWork".CoordSaldatura[8].X1;
_024: NOP   0;
      A     L 8.3;
      JNB   _025;
      L     "MD654";
      T     "DBWork".CoordSaldatura[8].Y1;
_025: NOP   0;
      A     L 8.2;
      AN    "DBWork".RotationTable;
      =     L 8.3;
      A     L 8.3;
      JNB   _026;
      L     "MD650";
      T     "DBWork".CoordSaldatura[8].X2;
_026: NOP   0;
      A     L 8.3;
      JNB   _027;
      L     "MD654";
      T     "DBWork".CoordSaldatura[8].Y2;
_027: NOP   0;
      A     L 8.1;
      A(;
      L     "DatiOP170B".PointWeldingTeachIn;
      L     9;
      ==I;
      );
      =     L 8.2;
      A     L 8.2;
      A     "DBWork".RotationTable;
      =     L 8.3;
      A     L 8.3;
      JNB   _028;
      L     "MD650";
      T     "DBWork".CoordSaldatura[9].X1;
_028: NOP   0;
      A     L 8.3;
      JNB   _029;
      L     "MD654";
      T     "DBWork".CoordSaldatura[9].Y1;
_029: NOP   0;
      A     L 8.2;
      AN    "DBWork".RotationTable;
      =     L 8.3;
      A     L 8.3;
      JNB   _02a;
      L     "MD650";
      T     "DBWork".CoordSaldatura[9].X2;
_02a: NOP   0;
      A     L 8.3;
      JNB   _02b;
      L     "MD654";
      T     "DBWork".CoordSaldatura[9].Y2;
_02b: NOP   0;
      A     L 8.1;
      A(;
      L     "DatiOP170B".PointWeldingTeachIn;
      L     10;
      ==I;
      );
      =     L 8.2;
      A     L 8.2;
      A     "DBWork".RotationTable;
      =     L 8.3;
      A     L 8.3;
      JNB   _02c;
      L     "MD650";
      T     "DBWork".CoordSaldatura[10].X1;
_02c: NOP   0;
      A     L 8.3;
      JNB   _02d;
      L     "MD654";
      T     "DBWork".CoordSaldatura[10].Y1;
_02d: NOP   0;
      A     L 8.2;
      AN    "DBWork".RotationTable;
      =     L 8.3;
      A     L 8.3;
      JNB   _02e;
      L     "MD650";
      T     "DBWork".CoordSaldatura[10].X2;
_02e: NOP   0;
      A     L 8.3;
      JNB   _02f;
      L     "MD654";
      T     "DBWork".CoordSaldatura[10].Y2;
_02f: NOP   0;
      A     L 8.1;
      A(;
      L     "DatiOP170B".PointWeldingTeachIn;
      L     11;
      ==I;
      );
      =     L 8.2;
      A     L 8.2;
      A     "DBWork".RotationTable;
      =     L 8.3;
      A     L 8.3;
      JNB   _030;
      L     "MD650";
      T     "DBWork".CoordSaldatura[11].X1;
_030: NOP   0;
      A     L 8.3;
      JNB   _031;
      L     "MD654";
      T     "DBWork".CoordSaldatura[11].Y1;
_031: NOP   0;
      A     L 8.2;
      AN    "DBWork".RotationTable;
      =     L 8.3;
      A     L 8.3;
      JNB   _032;
      L     "MD650";
      T     "DBWork".CoordSaldatura[11].X2;
_032: NOP   0;
      A     L 8.3;
      JNB   _033;
      L     "MD654";
      T     "DBWork".CoordSaldatura[11].Y2;
_033: NOP   0;
      A     L 8.1;
      A(;
      L     "DatiOP170B".PointWeldingTeachIn;
      L     12;
      ==I;
      );
      =     L 8.2;
      A     L 8.2;
      A     "DBWork".RotationTable;
      =     L 8.3;
      A     L 8.3;
      JNB   _034;
      L     "MD650";
      T     "DBWork".CoordSaldatura[12].X1;
_034: NOP   0;
      A     L 8.3;
      JNB   _035;
      L     "MD654";
      T     "DBWork".CoordSaldatura[12].Y1;
_035: NOP   0;
      A     L 8.2;
      AN    "DBWork".RotationTable;
      =     L 8.3;
      A     L 8.3;
      JNB   _036;
      L     "MD650";
      T     "DBWork".CoordSaldatura[12].X2;
_036: NOP   0;
      A     L 8.3;
      JNB   _037;
      L     "MD654";
      T     "DBWork".CoordSaldatura[12].Y2;
_037: NOP   0;
      A     L 8.1;
      A(;
      L     "DatiOP170B".PointWeldingTeachIn;
      L     13;
      ==I;
      );
      =     L 8.2;
      A     L 8.2;
      A     "DBWork".RotationTable;
      =     L 8.3;
      A     L 8.3;
      JNB   _038;
      L     "MD650";
      T     "DBWork".CoordSaldatura[13].X1;
_038: NOP   0;
      A     L 8.3;
      JNB   _039;
      L     "MD654";
      T     "DBWork".CoordSaldatura[13].Y1;
_039: NOP   0;
      A     L 8.2;
      AN    "DBWork".RotationTable;
      =     L 8.3;
      A     L 8.3;
      JNB   _03a;
      L     "MD650";
      T     "DBWork".CoordSaldatura[13].X2;
_03a: NOP   0;
      A     L 8.3;
      JNB   _03b;
      L     "MD654";
      T     "DBWork".CoordSaldatura[13].Y2;
_03b: NOP   0;
      A     L 8.1;
      A(;
      L     "DatiOP170B".PointWeldingTeachIn;
      L     14;
      ==I;
      );
      =     L 8.2;
      A     L 8.2;
      JNB   _03c;
      L     "MD650";
      T     "DBWork".STAT29[1].x;
_03c: NOP   0;
      A     L 8.2;
      JNB   _03d;
      L     "MD654";
      T     "DBWork".STAT29[1].y;
_03d: NOP   0;
      A     L 8.1;
      JNB   _03e;
      L     6;
      T     "DatiOP170B".PaginaDaVisualizzare;
_03e: NOP   0;
      A     L 8.1;
      JNB   _03f;
      L     "MD650";
      T     "MD588";
_03f: NOP   0;
      A     L 8.1;
      JNB   _040;
      L     "MD654";
      T     "MD592";
_040: NOP   0;
      A     L 8.1;
      BLD   102;
      S     "M75.1";
      A     L 8.1;
      FP    "M1004.5";
      JNB   _041;
      L     5;
      T     "DatiOP170B".PaginaDaVisualizzare;
_041: NOP   0;
      A     L 8.0;
      BLD   102;
      R     "M75.0";
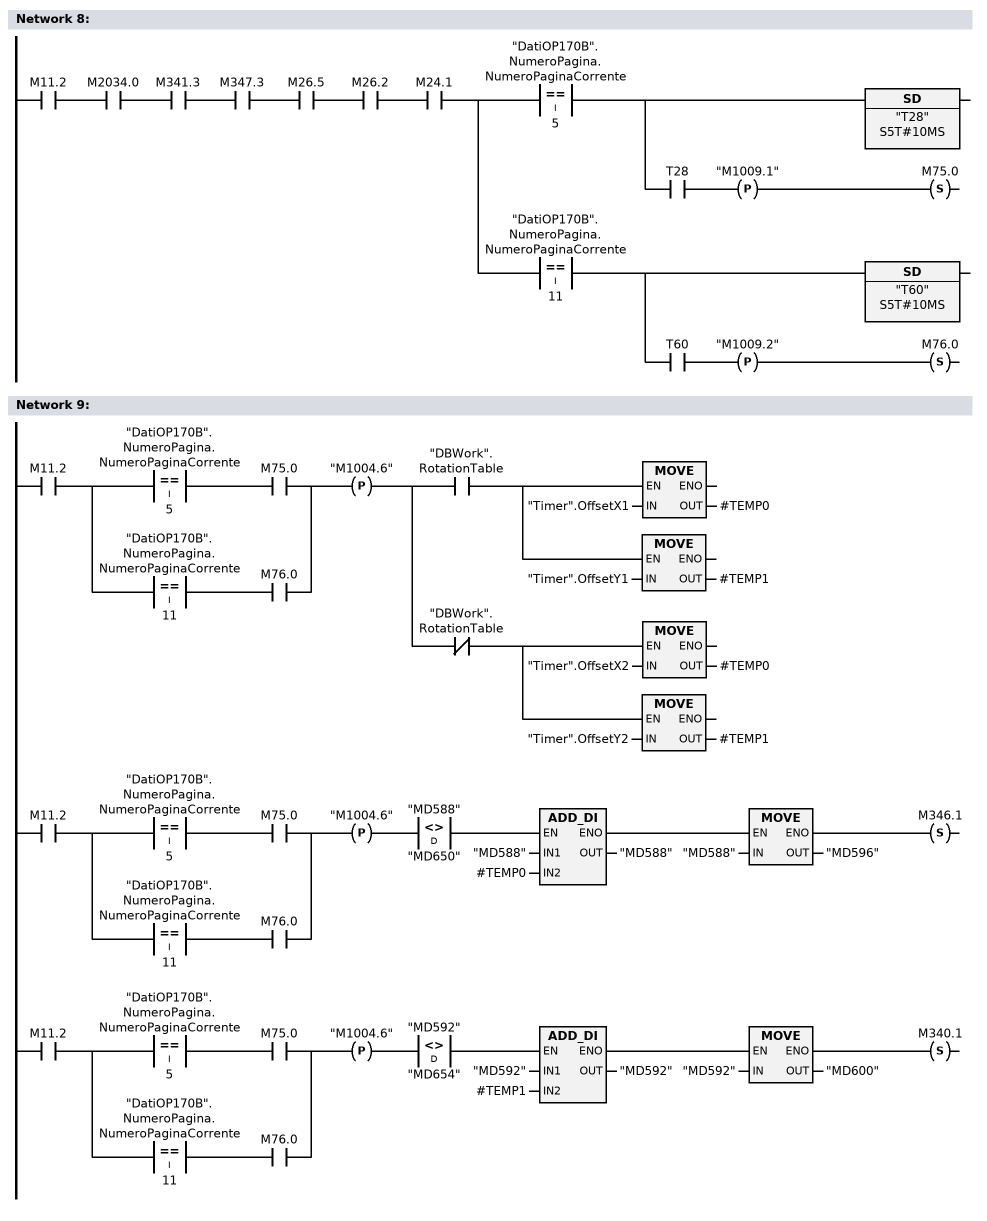
NETWORK
TITLE =
      A     "M11.2";
      A     "M2034.0";
      A     "M341.3";
      A     "M347.3";
      A     "M26.5";
      A     "M26.2";
      A     "M24.1";
      =     L 8.0;
      A     L 8.0;
      A(;
      L     "DatiOP170B".NumeroPagina.NumeroPaginaCorrente;
      L     5;
      ==I;
      );
      =     L 8.1;
      A     L 8.1;
      BLD   102;
      L     S5T#10MS;
      SD    "T28";
      A     L 8.1;
      A     "T28";
      FP    "M1009.1";
      S     "M75.0";
      A     L 8.0;
      A(;
      L     "DatiOP170B".NumeroPagina.NumeroPaginaCorrente;
      L     11;
      ==I;
      );
      =     L 8.1;
      A     L 8.1;
      BLD   102;
      L     S5T#10MS;
      SD    "T60";
      A     L 8.1;
      A     "T60";
      FP    "M1009.2";
      S     "M76.0";
NETWORK
TITLE =
      A     "M11.2";
      A(;
      A(;
      L     "DatiOP170B".NumeroPagina.NumeroPaginaCorrente;
      L     5;
      ==I;
      );
      A     "M75.0";
      O;
      A(;
      L     "DatiOP170B".NumeroPagina.NumeroPaginaCorrente;
      L     11;
      ==I;
      );
      A     "M76.0";
      );
      FP    "M1004.6";
      =     L 8.0;
      A     L 8.0;
      A     "DBWork".RotationTable;
      =     L 8.1;
      A     L 8.1;
      JNB   _042;
      L     "Timer".OffsetX1;
      T     #TEMP0;
_042: NOP   0;
      A     L 8.1;
      JNB   _043;
      L     "Timer".OffsetY1;
      T     #TEMP1;
_043: NOP   0;
      A     L 8.0;
      AN    "DBWork".RotationTable;
      =     L 8.1;
      A     L 8.1;
      JNB   _044;
      L     "Timer".OffsetX2;
      T     #TEMP0;
_044: NOP   0;
      A     L 8.1;
      JNB   _045;
      L     "Timer".OffsetY2;
      T     #TEMP1;
_045: NOP   0;
      A(;
      A     L 8.0;
      A(;
      L     "MD588";
      L     "MD650";
      <>D;
      );
      JNB   _046;
      L     "MD588";
      L     #TEMP0;
      +D;
      T     "MD588";
      AN    OV;
      SAVE;
      CLR;
_046: A     BR;
      );
      JNB   _047;
      L     "MD588";
      T     "MD596";
      SET;
      SAVE;
      CLR;
_047: A     BR;
      S     "M346.1";
      A(;
      A     L 8.0;
      A(;
      L     "MD592";
      L     "MD654";
      <>D;
      );
      JNB   _048;
      L     "MD592";
      L     #TEMP1;
      +D;
      T     "MD592";
      AN    OV;
      SAVE;
      CLR;
_048: A     BR;
      );
      JNB   _049;
      L     "MD592";
      T     "MD600";
      SET;
      SAVE;
      CLR;
_049: A     BR;
      S     "M340.1";
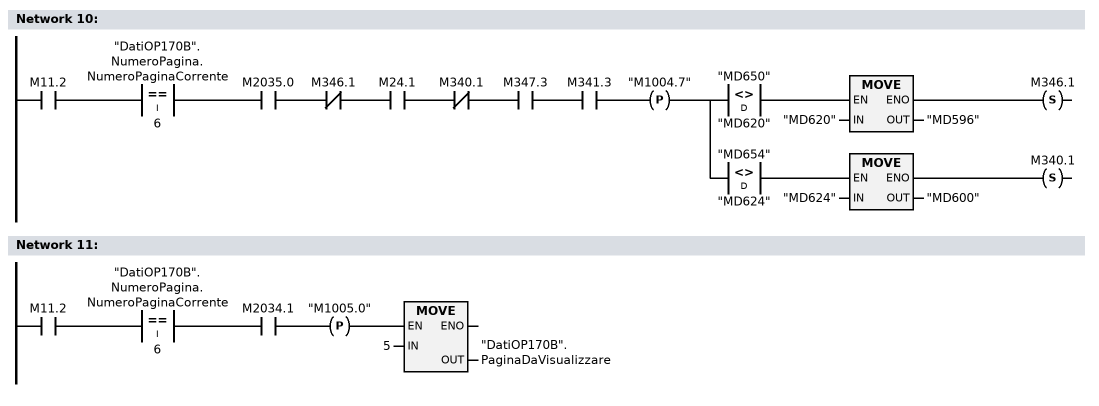
NETWORK
TITLE =
      A     "M11.2";
      A(;
      L     "DatiOP170B".NumeroPagina.NumeroPaginaCorrente;
      L     6;
      ==I;
      );
      A     "M2035.0";
      AN    "M346.1";
      A     "M24.1";
      AN    "M340.1";
      A     "M347.3";
      A     "M341.3";
      FP    "M1004.7";
      =     L 8.0;
      A     L 8.0;
      A(;
      L     "MD650";
      L     "MD620";
      <>D;
      );
      JNB   _04a;
      L     "MD620";
      T     "MD596";
      SET;
      SAVE;
      CLR;
_04a: A     BR;
      S     "M346.1";
      A     L 8.0;
      A(;
      L     "MD654";
      L     "MD624";
      <>D;
      );
      JNB   _04b;
      L     "MD624";
      T     "MD600";
      SET;
      SAVE;
      CLR;
_04b: A     BR;
      S     "M340.1";
NETWORK
TITLE =
      A     "M11.2";
      A(;
      L     "DatiOP170B".NumeroPagina.NumeroPaginaCorrente;
      L     6;
      ==I;
      );
      A     "M2034.1";
      FP    "M1005.0";
      JNB   _04c;
      L     5;
      T     "DatiOP170B".PaginaDaVisualizzare;
_04c: NOP   0;
END_FUNCTION

FUNCTION "FC51 - TYPE TOOL" : VOID	// FC 51
VERSION : 0.1
BEGIN
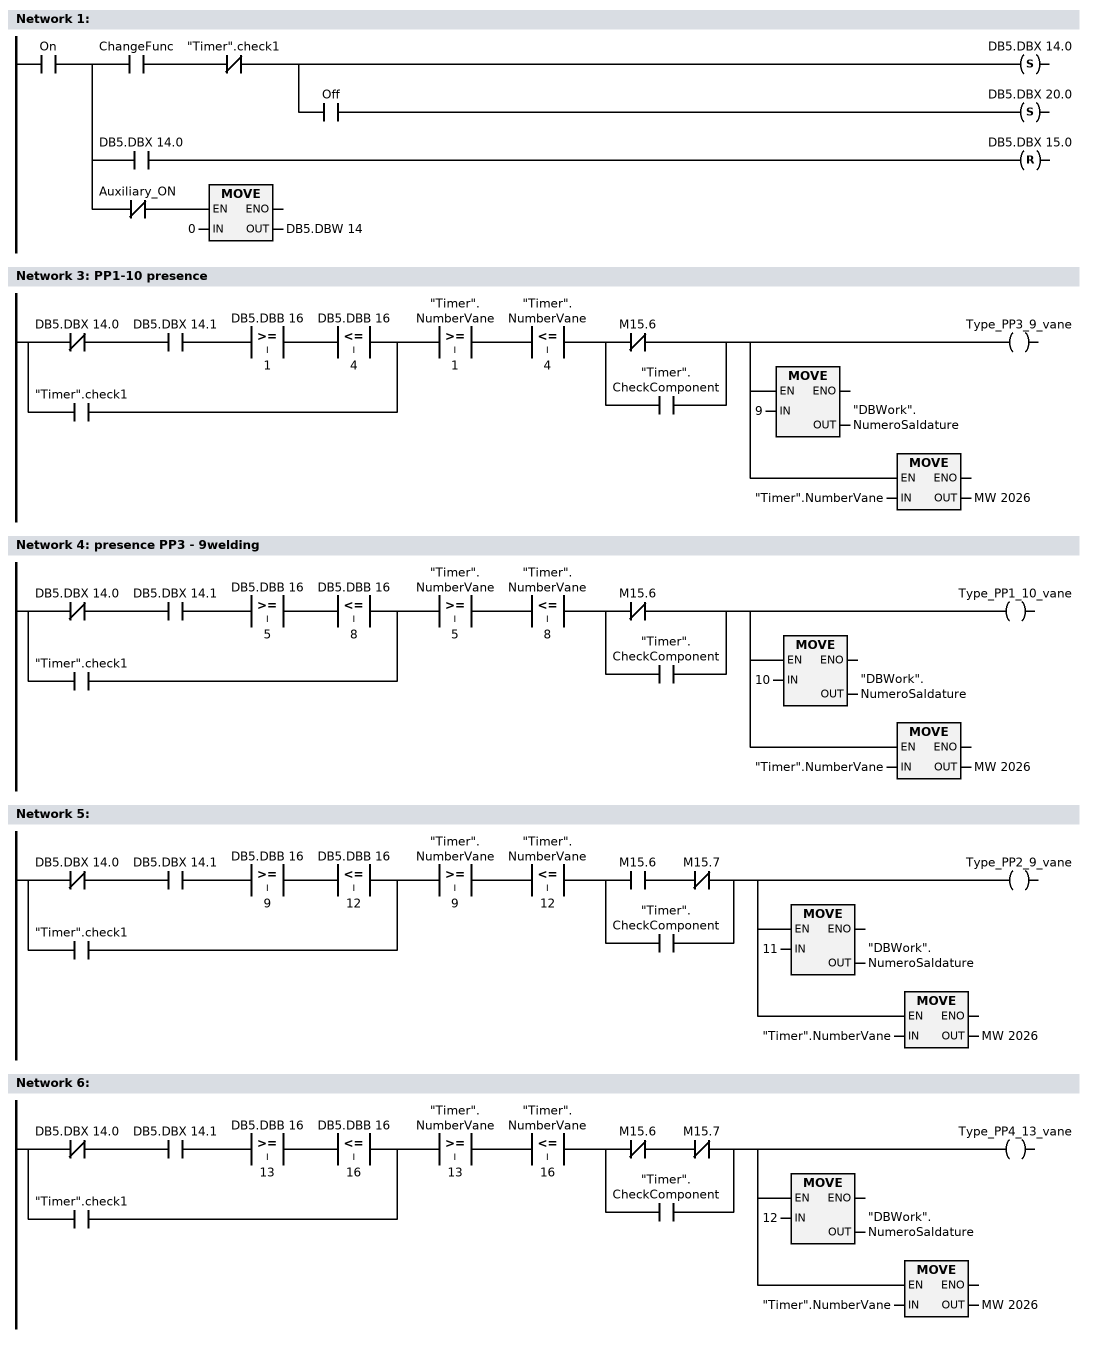
NETWORK
TITLE =
      A     "On";
      =     L 0.0;
      A     L 0.0;
      A     "ChangeFunc";
      AN    "Timer".check1;
      =     L 0.1;
      A     L 0.1;
      BLD   102;
      S     DB5.DBX 14.0;
      A     L 0.1;
      A     "Off";
      S     DB5.DBX 20.0;
      A     L 0.0;
      A     DB5.DBX 14.0;
      R     DB5.DBX 15.0;
      A     L 0.0;
      AN    "Auxiliary_ON";
      JNB   _001;
      L     0;
      T     DB5.DBW 14;
_001: NOP   0;
NETWORK
TITLE =
NETWORK
TITLE = PP1-10 presence
      A(;
      AN    DB5.DBX 14.0;
      A     DB5.DBX 14.1;
      A(;
      L     DB5.DBB 16;
      L     1;
      >=I;
      );
      A(;
      L     DB5.DBB 16;
      L     4;
      <=I;
      );
      O     "Timer".check1;
      );
      A(;
      L     "Timer".NumberVane;
      L     1;
      >=I;
      );
      A(;
      L     "Timer".NumberVane;
      L     4;
      <=I;
      );
      A(;
      ON    "M15.6";
      O     "Timer".CheckComponent;
      );
      =     L 0.0;
      A     L 0.0;
      BLD   102;
      =     "Type_PP3_9_vane";
      A     L 0.0;
      JNB   _002;
      L     9;
      T     "DBWork".NumeroSaldature;
_002: NOP   0;
      A     L 0.0;
      JNB   _003;
      L     "Timer".NumberVane;
      T     MW 2026;
_003: NOP   0;
NETWORK
TITLE = presence PP3 - 9welding
      A(;
      AN    DB5.DBX 14.0;
      A     DB5.DBX 14.1;
      A(;
      L     DB5.DBB 16;
      L     5;
      >=I;
      );
      A(;
      L     DB5.DBB 16;
      L     8;
      <=I;
      );
      O     "Timer".check1;
      );
      A(;
      L     "Timer".NumberVane;
      L     5;
      >=I;
      );
      A(;
      L     "Timer".NumberVane;
      L     8;
      <=I;
      );
      A(;
      ON    "M15.6";
      O     "Timer".CheckComponent;
      );
      =     L 0.0;
      A     L 0.0;
      BLD   102;
      =     "Type_PP1_10_vane";
      A     L 0.0;
      JNB   _004;
      L     10;
      T     "DBWork".NumeroSaldature;
_004: NOP   0;
      A     L 0.0;
      JNB   _005;
      L     "Timer".NumberVane;
      T     MW 2026;
_005: NOP   0;
NETWORK
TITLE =
      A(;
      AN    DB5.DBX 14.0;
      A     DB5.DBX 14.1;
      A(;
      L     DB5.DBB 16;
      L     9;
      >=I;
      );
      A(;
      L     DB5.DBB 16;
      L     12;
      <=I;
      );
      O     "Timer".check1;
      );
      A(;
      L     "Timer".NumberVane;
      L     9;
      >=I;
      );
      A(;
      L     "Timer".NumberVane;
      L     12;
      <=I;
      );
      A(;
      A     "M15.6";
      AN    "M15.7";
      O     "Timer".CheckComponent;
      );
      =     L 0.0;
      A     L 0.0;
      BLD   102;
      =     "Type_PP2_9_vane";
      A     L 0.0;
      JNB   _006;
      L     11;
      T     "DBWork".NumeroSaldature;
_006: NOP   0;
      A     L 0.0;
      JNB   _007;
      L     "Timer".NumberVane;
      T     MW 2026;
_007: NOP   0;
NETWORK
TITLE =
      A(;
      AN    DB5.DBX 14.0;
      A     DB5.DBX 14.1;
      A(;
      L     DB5.DBB 16;
      L     13;
      >=I;
      );
      A(;
      L     DB5.DBB 16;
      L     16;
      <=I;
      );
      O     "Timer".check1;
      );
      A(;
      L     "Timer".NumberVane;
      L     13;
      >=I;
      );
      A(;
      L     "Timer".NumberVane;
      L     16;
      <=I;
      );
      A(;
      AN    "M15.6";
      AN    "M15.7";
      O     "Timer".CheckComponent;
      );
      =     L 0.0;
      A     L 0.0;
      BLD   102;
      =     "Type_PP4_13_vane";
      A     L 0.0;
      JNB   _008;
      L     12;
      T     "DBWork".NumeroSaldature;
_008: NOP   0;
      A     L 0.0;
      JNB   _009;
      L     "Timer".NumberVane;
      T     MW 2026;
_009: NOP   0;
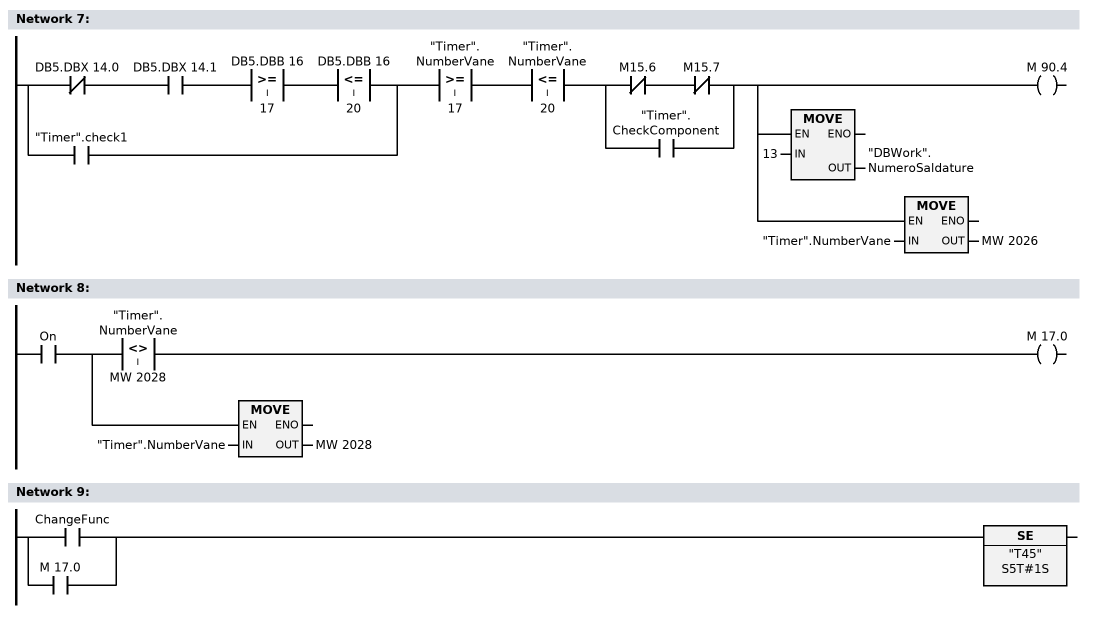
NETWORK
TITLE =
      A(;
      AN    DB5.DBX 14.0;
      A     DB5.DBX 14.1;
      A(;
      L     DB5.DBB 16;
      L     17;
      >=I;
      );
      A(;
      L     DB5.DBB 16;
      L     20;
      <=I;
      );
      O     "Timer".check1;
      );
      A(;
      L     "Timer".NumberVane;
      L     17;
      >=I;
      );
      A(;
      L     "Timer".NumberVane;
      L     20;
      <=I;
      );
      A(;
      AN    "M15.6";
      AN    "M15.7";
      O     "Timer".CheckComponent;
      );
      =     L 0.0;
      A     L 0.0;
      BLD   102;
      =     M 90.4;
      A     L 0.0;
      JNB   _00a;
      L     13;
      T     "DBWork".NumeroSaldature;
_00a: NOP   0;
      A     L 0.0;
      JNB   _00b;
      L     "Timer".NumberVane;
      T     MW 2026;
_00b: NOP   0;
NETWORK
TITLE =
      A     "On";
      =     L 0.0;
      A     L 0.0;
      A(;
      L     "Timer".NumberVane;
      L     MW 2028;
      <>I;
      );
      =     M 17.0;
      A     L 0.0;
      JNB   _00c;
      L     "Timer".NumberVane;
      T     MW 2028;
_00c: NOP   0;
NETWORK
TITLE =
      O     "ChangeFunc";
      O     M 17.0;
      L     S5T#1S;
      SE    "T45";
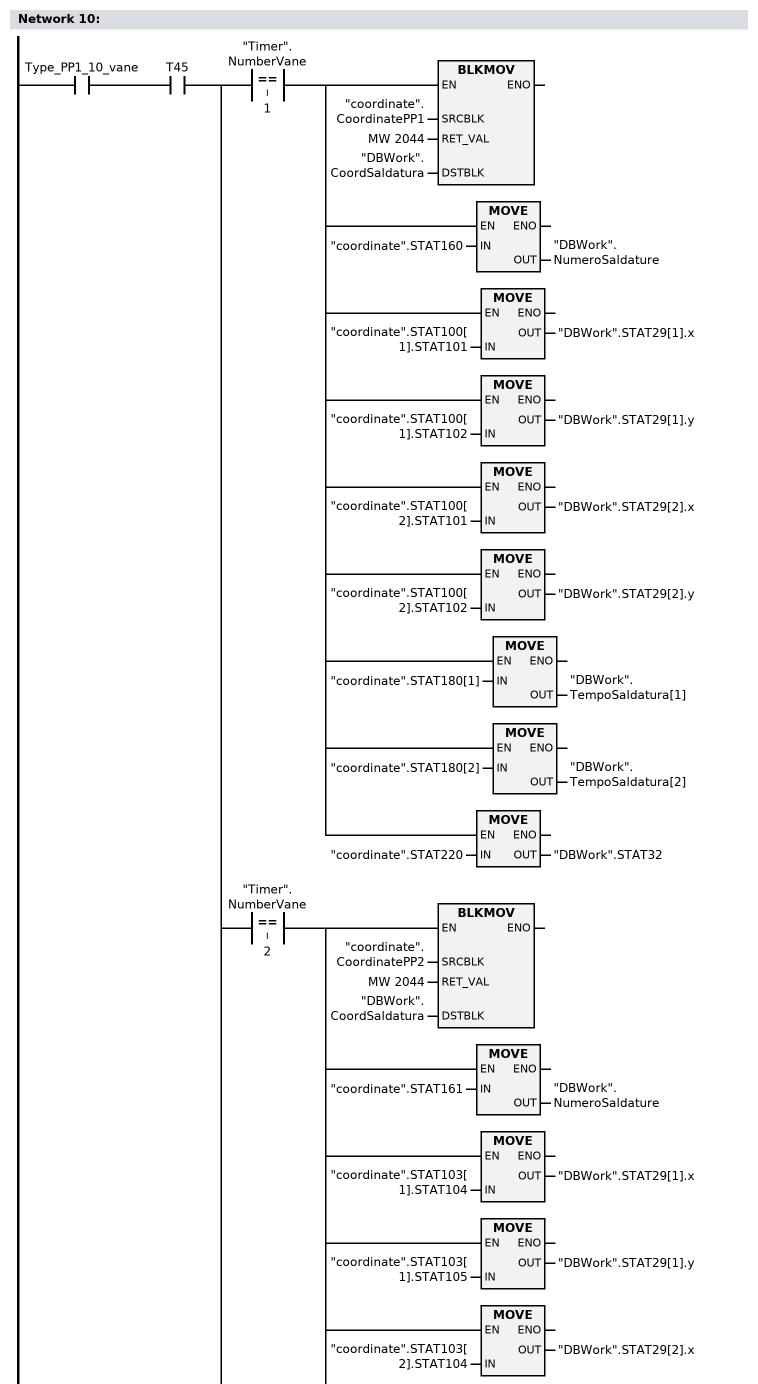
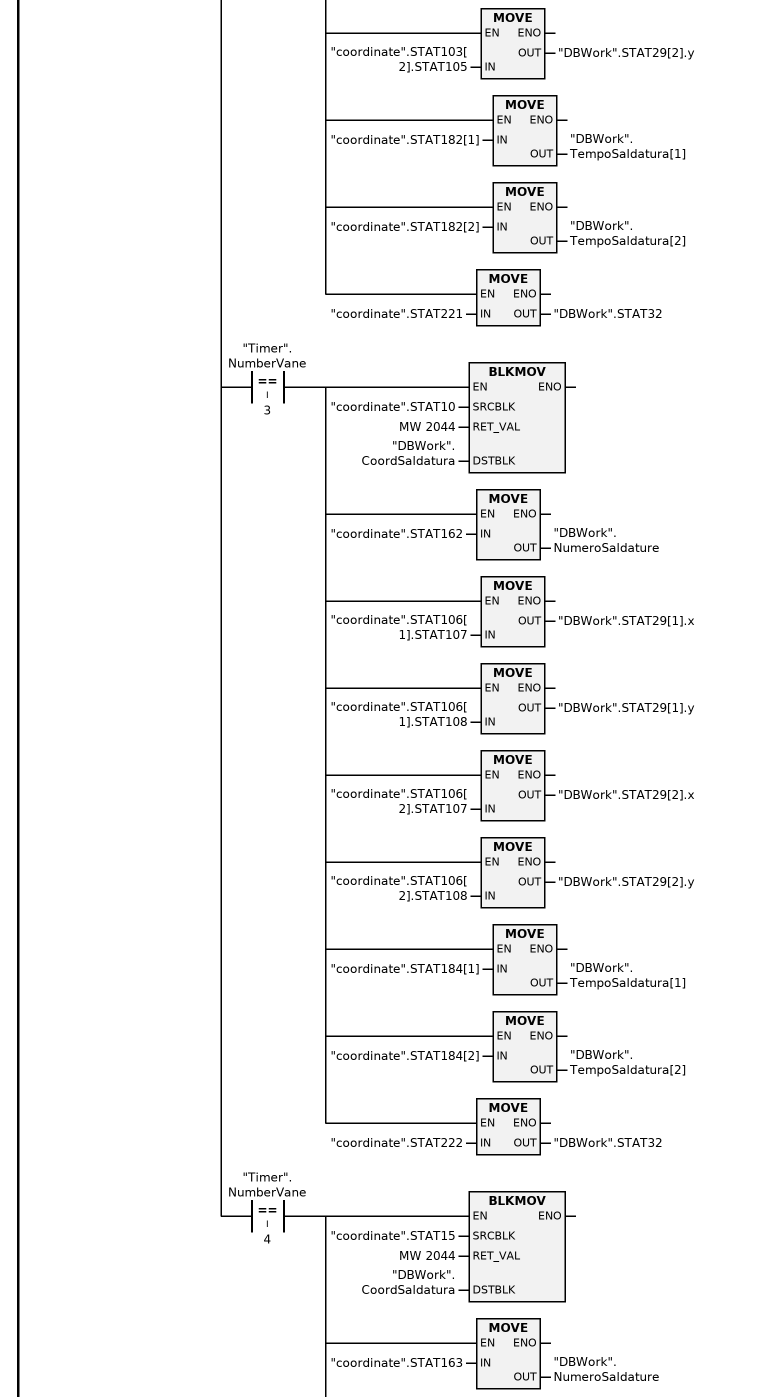
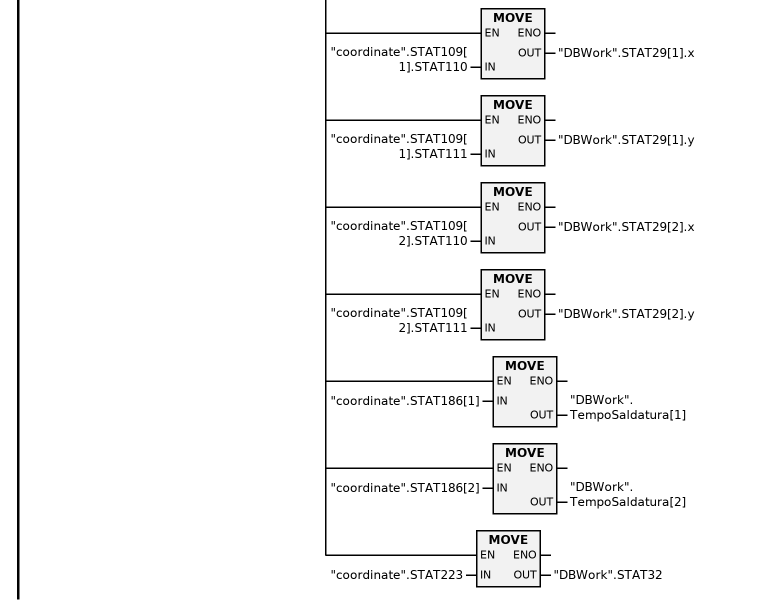
NETWORK
TITLE =
      A     "Type_PP1_10_vane";
      A     "T45";
      =     L 0.0;
      A     L 0.0;
      A(;
      L     "Timer".NumberVane;
      L     1;
      ==I;
      );
      =     L 0.1;
      A     L 0.1;
      JNB   _00d;
      CALL  "BLKMOV" (
           SRCBLK                   := "coordinate".CoordinatePP1,
           RET_VAL                  := MW 2044,
           DSTBLK                   := "DBWork".CoordSaldatura);
_00d: NOP   0;
      A     L 0.1;
      JNB   _00e;
      L     "coordinate".STAT160;
      T     "DBWork".NumeroSaldature;
_00e: NOP   0;
      A     L 0.1;
      JNB   _00f;
      L     "coordinate".STAT100[1].STAT101;
      T     "DBWork".STAT29[1].x;
_00f: NOP   0;
      A     L 0.1;
      JNB   _010;
      L     "coordinate".STAT100[1].STAT102;
      T     "DBWork".STAT29[1].y;
_010: NOP   0;
      A     L 0.1;
      JNB   _011;
      L     "coordinate".STAT100[2].STAT101;
      T     "DBWork".STAT29[2].x;
_011: NOP   0;
      A     L 0.1;
      JNB   _012;
      L     "coordinate".STAT100[2].STAT102;
      T     "DBWork".STAT29[2].y;
_012: NOP   0;
      A     L 0.1;
      JNB   _013;
      L     "coordinate".STAT180[1];
      T     "DBWork".TempoSaldatura[1];
_013: NOP   0;
      A     L 0.1;
      JNB   _014;
      L     "coordinate".STAT180[2];
      T     "DBWork".TempoSaldatura[2];
_014: NOP   0;
      A     L 0.1;
      JNB   _015;
      L     "coordinate".STAT220;
      T     "DBWork".STAT32;
_015: NOP   0;
      A     L 0.0;
      A(;
      L     "Timer".NumberVane;
      L     2;
      ==I;
      );
      =     L 0.1;
      A     L 0.1;
      JNB   _016;
      CALL  "BLKMOV" (
           SRCBLK                   := "coordinate".CoordinatePP2,
           RET_VAL                  := MW 2044,
           DSTBLK                   := "DBWork".CoordSaldatura);
_016: NOP   0;
      A     L 0.1;
      JNB   _017;
      L     "coordinate".STAT161;
      T     "DBWork".NumeroSaldature;
_017: NOP   0;
      A     L 0.1;
      JNB   _018;
      L     "coordinate".STAT103[1].STAT104;
      T     "DBWork".STAT29[1].x;
_018: NOP   0;
      A     L 0.1;
      JNB   _019;
      L     "coordinate".STAT103[1].STAT105;
      T     "DBWork".STAT29[1].y;
_019: NOP   0;
      A     L 0.1;
      JNB   _01a;
      L     "coordinate".STAT103[2].STAT104;
      T     "DBWork".STAT29[2].x;
_01a: NOP   0;
      A     L 0.1;
      JNB   _01b;
      L     "coordinate".STAT103[2].STAT105;
      T     "DBWork".STAT29[2].y;
_01b: NOP   0;
      A     L 0.1;
      JNB   _01c;
      L     "coordinate".STAT182[1];
      T     "DBWork".TempoSaldatura[1];
_01c: NOP   0;
      A     L 0.1;
      JNB   _01d;
      L     "coordinate".STAT182[2];
      T     "DBWork".TempoSaldatura[2];
_01d: NOP   0;
      A     L 0.1;
      JNB   _01e;
      L     "coordinate".STAT221;
      T     "DBWork".STAT32;
_01e: NOP   0;
      A     L 0.0;
      A(;
      L     "Timer".NumberVane;
      L     3;
      ==I;
      );
      =     L 0.1;
      A     L 0.1;
      JNB   _01f;
      CALL  "BLKMOV" (
           SRCBLK                   := "coordinate".STAT10,
           RET_VAL                  := MW 2044,
           DSTBLK                   := "DBWork".CoordSaldatura);
_01f: NOP   0;
      A     L 0.1;
      JNB   _020;
      L     "coordinate".STAT162;
      T     "DBWork".NumeroSaldature;
_020: NOP   0;
      A     L 0.1;
      JNB   _021;
      L     "coordinate".STAT106[1].STAT107;
      T     "DBWork".STAT29[1].x;
_021: NOP   0;
      A     L 0.1;
      JNB   _022;
      L     "coordinate".STAT106[1].STAT108;
      T     "DBWork".STAT29[1].y;
_022: NOP   0;
      A     L 0.1;
      JNB   _023;
      L     "coordinate".STAT106[2].STAT107;
      T     "DBWork".STAT29[2].x;
_023: NOP   0;
      A     L 0.1;
      JNB   _024;
      L     "coordinate".STAT106[2].STAT108;
      T     "DBWork".STAT29[2].y;
_024: NOP   0;
      A     L 0.1;
      JNB   _025;
      L     "coordinate".STAT184[1];
      T     "DBWork".TempoSaldatura[1];
_025: NOP   0;
      A     L 0.1;
      JNB   _026;
      L     "coordinate".STAT184[2];
      T     "DBWork".TempoSaldatura[2];
_026: NOP   0;
      A     L 0.1;
      JNB   _027;
      L     "coordinate".STAT222;
      T     "DBWork".STAT32;
_027: NOP   0;
      A     L 0.0;
      A(;
      L     "Timer".NumberVane;
      L     4;
      ==I;
      );
      =     L 0.1;
      A     L 0.1;
      JNB   _028;
      CALL  "BLKMOV" (
           SRCBLK                   := "coordinate".STAT15,
           RET_VAL                  := MW 2044,
           DSTBLK                   := "DBWork".CoordSaldatura);
_028: NOP   0;
      A     L 0.1;
      JNB   _029;
      L     "coordinate".STAT163;
      T     "DBWork".NumeroSaldature;
_029: NOP   0;
      A     L 0.1;
      JNB   _02a;
      L     "coordinate".STAT109[1].STAT110;
      T     "DBWork".STAT29[1].x;
_02a: NOP   0;
      A     L 0.1;
      JNB   _02b;
      L     "coordinate".STAT109[1].STAT111;
      T     "DBWork".STAT29[1].y;
_02b: NOP   0;
      A     L 0.1;
      JNB   _02c;
      L     "coordinate".STAT109[2].STAT110;
      T     "DBWork".STAT29[2].x;
_02c: NOP   0;
      A     L 0.1;
      JNB   _02d;
      L     "coordinate".STAT109[2].STAT111;
      T     "DBWork".STAT29[2].y;
_02d: NOP   0;
      A     L 0.1;
      JNB   _02e;
      L     "coordinate".STAT186[1];
      T     "DBWork".TempoSaldatura[1];
_02e: NOP   0;
      A     L 0.1;
      JNB   _02f;
      L     "coordinate".STAT186[2];
      T     "DBWork".TempoSaldatura[2];
_02f: NOP   0;
      A     L 0.1;
      JNB   _030;
      L     "coordinate".STAT223;
      T     "DBWork".STAT32;
_030: NOP   0;
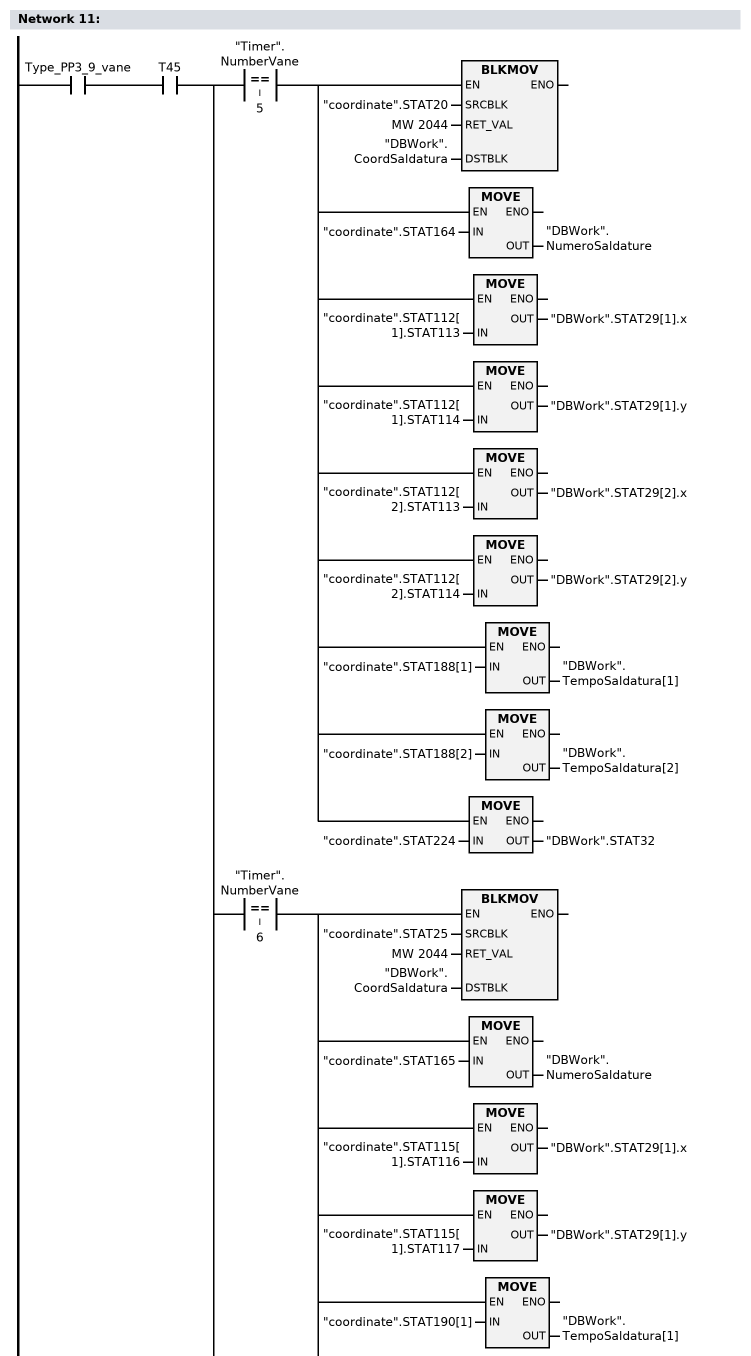
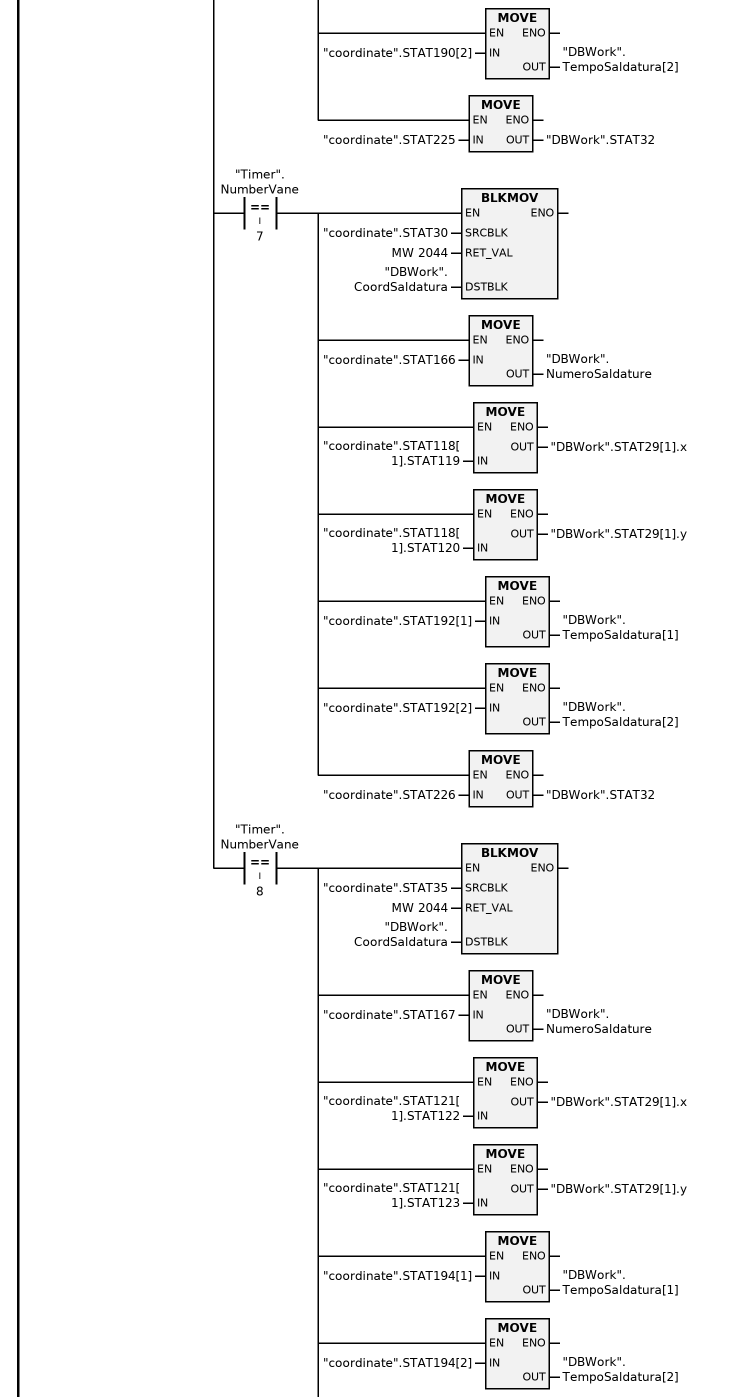
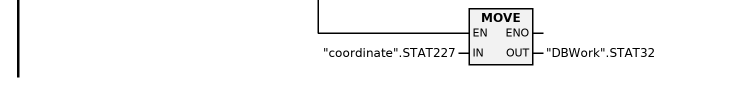
NETWORK
TITLE =
      A     "Type_PP3_9_vane";
      A     "T45";
      =     L 0.0;
      A     L 0.0;
      A(;
      L     "Timer".NumberVane;
      L     5;
      ==I;
      );
      =     L 0.1;
      A     L 0.1;
      JNB   _031;
      CALL  "BLKMOV" (
           SRCBLK                   := "coordinate".STAT20,
           RET_VAL                  := MW 2044,
           DSTBLK                   := "DBWork".CoordSaldatura);
_031: NOP   0;
      A     L 0.1;
      JNB   _032;
      L     "coordinate".STAT164;
      T     "DBWork".NumeroSaldature;
_032: NOP   0;
      A     L 0.1;
      JNB   _033;
      L     "coordinate".STAT112[1].STAT113;
      T     "DBWork".STAT29[1].x;
_033: NOP   0;
      A     L 0.1;
      JNB   _034;
      L     "coordinate".STAT112[1].STAT114;
      T     "DBWork".STAT29[1].y;
_034: NOP   0;
      A     L 0.1;
      JNB   _035;
      L     "coordinate".STAT112[2].STAT113;
      T     "DBWork".STAT29[2].x;
_035: NOP   0;
      A     L 0.1;
      JNB   _036;
      L     "coordinate".STAT112[2].STAT114;
      T     "DBWork".STAT29[2].y;
_036: NOP   0;
      A     L 0.1;
      JNB   _037;
      L     "coordinate".STAT188[1];
      T     "DBWork".TempoSaldatura[1];
_037: NOP   0;
      A     L 0.1;
      JNB   _038;
      L     "coordinate".STAT188[2];
      T     "DBWork".TempoSaldatura[2];
_038: NOP   0;
      A     L 0.1;
      JNB   _039;
      L     "coordinate".STAT224;
      T     "DBWork".STAT32;
_039: NOP   0;
      A     L 0.0;
      A(;
      L     "Timer".NumberVane;
      L     6;
      ==I;
      );
      =     L 0.1;
      A     L 0.1;
      JNB   _03a;
      CALL  "BLKMOV" (
           SRCBLK                   := "coordinate".STAT25,
           RET_VAL                  := MW 2044,
           DSTBLK                   := "DBWork".CoordSaldatura);
_03a: NOP   0;
      A     L 0.1;
      JNB   _03b;
      L     "coordinate".STAT165;
      T     "DBWork".NumeroSaldature;
_03b: NOP   0;
      A     L 0.1;
      JNB   _03c;
      L     "coordinate".STAT115[1].STAT116;
      T     "DBWork".STAT29[1].x;
_03c: NOP   0;
      A     L 0.1;
      JNB   _03d;
      L     "coordinate".STAT115[1].STAT117;
      T     "DBWork".STAT29[1].y;
_03d: NOP   0;
      A     L 0.1;
      JNB   _03e;
      L     "coordinate".STAT190[1];
      T     "DBWork".TempoSaldatura[1];
_03e: NOP   0;
      A     L 0.1;
      JNB   _03f;
      L     "coordinate".STAT190[2];
      T     "DBWork".TempoSaldatura[2];
_03f: NOP   0;
      A     L 0.1;
      JNB   _040;
      L     "coordinate".STAT225;
      T     "DBWork".STAT32;
_040: NOP   0;
      A     L 0.0;
      A(;
      L     "Timer".NumberVane;
      L     7;
      ==I;
      );
      =     L 0.1;
      A     L 0.1;
      JNB   _041;
      CALL  "BLKMOV" (
           SRCBLK                   := "coordinate".STAT30,
           RET_VAL                  := MW 2044,
           DSTBLK                   := "DBWork".CoordSaldatura);
_041: NOP   0;
      A     L 0.1;
      JNB   _042;
      L     "coordinate".STAT166;
      T     "DBWork".NumeroSaldature;
_042: NOP   0;
      A     L 0.1;
      JNB   _043;
      L     "coordinate".STAT118[1].STAT119;
      T     "DBWork".STAT29[1].x;
_043: NOP   0;
      A     L 0.1;
      JNB   _044;
      L     "coordinate".STAT118[1].STAT120;
      T     "DBWork".STAT29[1].y;
_044: NOP   0;
      A     L 0.1;
      JNB   _045;
      L     "coordinate".STAT192[1];
      T     "DBWork".TempoSaldatura[1];
_045: NOP   0;
      A     L 0.1;
      JNB   _046;
      L     "coordinate".STAT192[2];
      T     "DBWork".TempoSaldatura[2];
_046: NOP   0;
      A     L 0.1;
      JNB   _047;
      L     "coordinate".STAT226;
      T     "DBWork".STAT32;
_047: NOP   0;
      A     L 0.0;
      A(;
      L     "Timer".NumberVane;
      L     8;
      ==I;
      );
      =     L 0.1;
      A     L 0.1;
      JNB   _048;
      CALL  "BLKMOV" (
           SRCBLK                   := "coordinate".STAT35,
           RET_VAL                  := MW 2044,
           DSTBLK                   := "DBWork".CoordSaldatura);
_048: NOP   0;
      A     L 0.1;
      JNB   _049;
      L     "coordinate".STAT167;
      T     "DBWork".NumeroSaldature;
_049: NOP   0;
      A     L 0.1;
      JNB   _04a;
      L     "coordinate".STAT121[1].STAT122;
      T     "DBWork".STAT29[1].x;
_04a: NOP   0;
      A     L 0.1;
      JNB   _04b;
      L     "coordinate".STAT121[1].STAT123;
      T     "DBWork".STAT29[1].y;
_04b: NOP   0;
      A     L 0.1;
      JNB   _04c;
      L     "coordinate".STAT194[1];
      T     "DBWork".TempoSaldatura[1];
_04c: NOP   0;
      A     L 0.1;
      JNB   _04d;
      L     "coordinate".STAT194[2];
      T     "DBWork".TempoSaldatura[2];
_04d: NOP   0;
      A     L 0.1;
      JNB   _04e;
      L     "coordinate".STAT227;
      T     "DBWork".STAT32;
_04e: NOP   0;
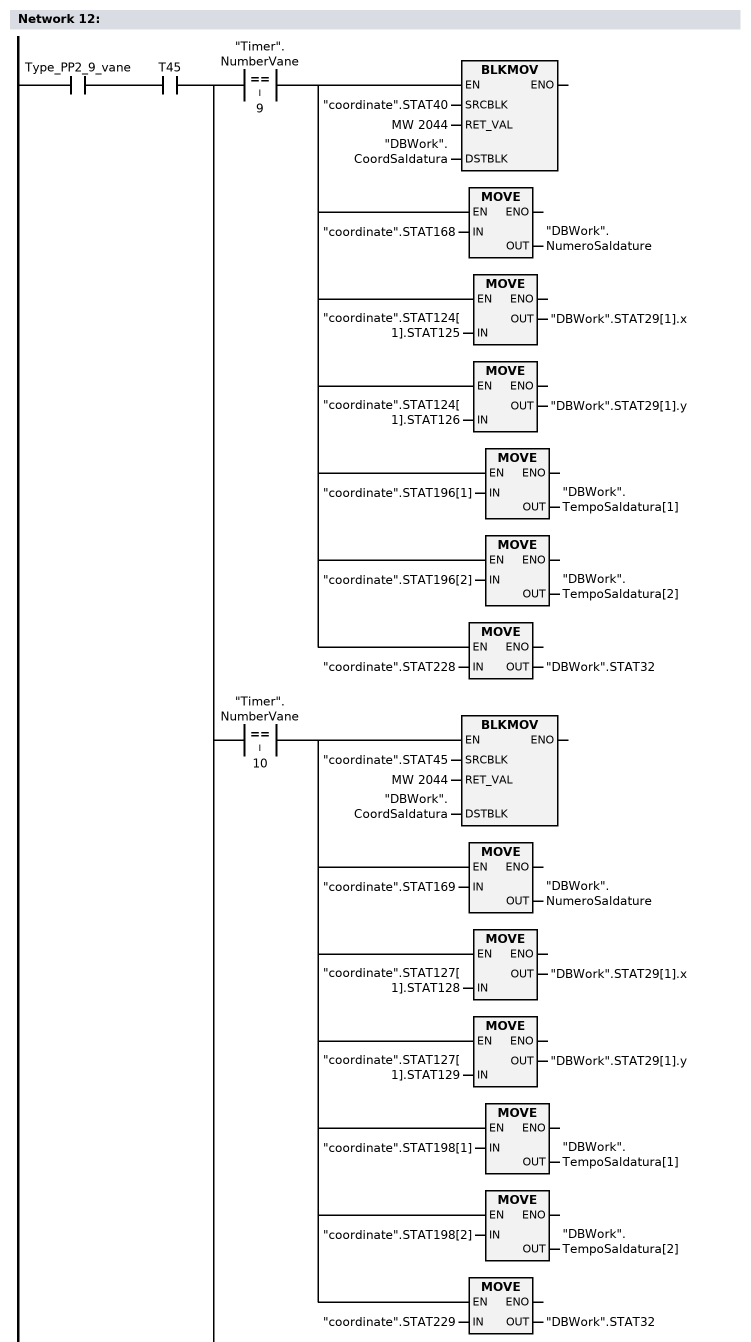
